COMM SMOVL C00426 BC00426 V=11.7  +MOVJ EC00426
COMM SMOVL C00427 BC00427 V=11.7  +MOVJ EC00427
COMM SFTON3D P062
COMM SMOVL C00428 BC00428 V=11.0  +MOVJ EC00428
COMM SMOVL C00429 BC00429 V=11.0  +MOVJ EC00429
COMM SFTON3D P061
COMM SMOVL C00430 BC00430 V=11.0  +MOVJ EC00430
COMM SMOVL C00431 BC00431 V=11.0  +MOVJ EC00431
COMM ARCOF
COMM SMOVL C00432 BC00432 V=800.0  +MOVJ EC00432
COMM SFTOF3D
COMM MOVJ C00433 BC00433 VJ=80.00  +MOVJ EC00433 VJ=80.00
COMM MOVJ C00434 BC00434 VJ=80.00  +MOVJ EC00434 VJ=80.00
COMM MOVJ C00435 BC00435 VJ=80.00  +MOVJ EC00435 VJ=80.00
COMM 'EndPath W3485
COMM 'Path W3486
COMM SFTOF3D
COMM SFTON3D P050
COMM MOVJ C00436 BC00436 VJ=100.00  +MOVJ EC00436 VJ=100.00
COMM SMOVL C00437 BC00437 V=800.0  +MOVJ EC00437
COMM SMOVL C00438 BC00438 V=150.0 PL=0  +MOVJ EC00438
COMM MACRO1 MJ#(0) ARGF14
COMM ARCON
COMM SMOVL C00439 BC00439 V=10.0  +MOVJ EC00439
COMM SMOVL C00440 BC00440 V=10.0  +MOVJ EC00440
COMM SMOVL C00441 BC00441 V=10.0  +MOVJ EC00441
COMM ARCOF
COMM SMOVL C00442 BC00442 V=800.0  +MOVJ EC00442
COMM SMOVL C00443 BC00443 V=1000.0  +MOVJ EC00443
COMM SFTOF3D
COMM 'EndPath W3486
COMM MOVJ C00444 BC00444 VJ=100.00  +MOVJ EC00444 VJ=100.00
COMM 'Path W3485
COMM SFTOF3D
COMM SFTON3D P034
COMM MOVJ C00445 BC00445 VJ=100.00  +MOVJ EC00445 VJ=100.00
COMM SMOVL C00446 BC00446 V=800.0  +MOVJ EC00446
COMM SMOVL C00447 BC00447 V=166.7 PL=0  +MOVJ EC00447
COMM ARCON
COMM SMOVL C00448 BC00448 V=9.2  +MOVJ EC00448
COMM SMOVL C00449 BC00449 V=9.2  +MOVJ EC00449
COMM SMOVL C00450 BC00450 V=9.2  +MOVJ EC00450
COMM ARCOF
COMM SMOVL C00451 BC00451 V=800.0  +MOVJ EC00451
COMM SMOVL C00452 BC00452 V=1000.0  +MOVJ EC00452
COMM SFTOF3D
COMM 'EndPath W3485
COMM 'Path W3487
COMM SFTOF3D
COMM SFTON3D P054
COMM MOVJ C00453 BC00453 VJ=100.00  +MOVJ EC00453 VJ=100.00
COMM SMOVL C00454 BC00454 V=800.0  +MOVJ EC00454
COMM SMOVL C00455 BC00455 V=150.0 PL=0  +MOVJ EC00455
COMM ARCON
COMM SMOVL C00456 BC00456 V=9.2  +MOVJ EC00456
COMM SMOVL C00457 BC00457 V=9.2  +MOVJ EC00457
COMM SMOVL C00458 BC00458 V=9.2  +MOVJ EC00458
COMM ARCOF
COMM SMOVL C00459 BC00459 V=800.0  +MOVJ EC00459
COMM SMOVL C00460 BC00460 V=1000.0  +MOVJ EC00460
COMM SFTOF3D
COMM 'EndPath W3487
COMM MOVJ C00461 BC00461 VJ=100.00  +MOVJ EC00461 VJ=100.00
COMM 'Path W3487
COMM SFTOF3D
COMM SFTON3D P028
COMM MOVJ C00462 BC00462 VJ=100.00  +MOVJ EC00462 VJ=100.00
COMM SMOVL C00463 BC00463 V=800.0  +MOVJ EC00463
COMM SMOVL C00464 BC00464 V=150.0 PL=0  +MOVJ EC00464
COMM ARCON
COMM SMOVL C00465 BC00465 V=9.2  +MOVJ EC00465
COMM SMOVL C00466 BC00466 V=9.2  +MOVJ EC00466
COMM SMOVL C00467 BC00467 V=9.2  +MOVJ EC00467
COMM ARCOF
COMM SMOVL C00468 BC00468 V=800.0  +MOVJ EC00468
COMM SMOVL C00469 BC00469 V=1000.0  +MOVJ EC00469
COMM SFTOF3D
COMM 'EndPath W3487
COMM MOVJ C00470 BC00470 VJ=100.00  +MOVJ EC00470 VJ=100.00
COMM MOVJ C00471 BC00471 VJ=100.00  +MOVJ EC00471 VJ=100.00
COMM 'brak dostepu offset 5mm
COMM 'Path W3488
COMM SFTOF3D
COMM SFTON3D P028
COMM MOVJ C00472 BC00472 VJ=100.00  +MOVJ EC00472 VJ=100.00
COMM SMOVL C00473 BC00473 V=800.0  +MOVJ EC00473
COMM SMOVL C00474 BC00474 V=150.0 PL=0  +MOVJ EC00474
COMM ARCON
COMM SMOVL C00475 BC00475 V=11.7  +MOVJ EC00475
COMM ARCOF
COMM SMOVL C00476 BC00476 V=800.0  +MOVJ EC00476
COMM SMOVL C00477 BC00477 V=1000.0  +MOVJ EC00477
COMM SFTOF3D
COMM 'EndPath W3488
COMM MOVJ C00478 BC00478 VJ=100.00  +MOVJ EC00478 VJ=100.00
COMM '13
COMM 'Path W3489
COMM SFTOF3D
COMM SFTON3D P030
COMM MOVJ C00479 BC00479 VJ=100.00  +MOVJ EC00479 VJ=100.00
COMM SMOVL C00480 BC00480 V=800.0  +MOVJ EC00480
COMM SMOVL C00481 BC00481 V=150.0 PL=0  +MOVJ EC00481
COMM MACRO1 MJ#(0) ARGF9
COMM ARCON
COMM SWVON WEV#(10)
COMM SFTON3D P031
COMM SMOVL C00482 BC00482 V=12.5  +MOVJ EC00482
COMM ARCOF
COMM SWVOF
COMM SMOVL C00483 BC00483 V=800.0  +MOVJ EC00483
COMM SMOVL C00484 BC00484 V=1000.0  +MOVJ EC00484
COMM SFTOF3D
COMM 'EndPath W3489
COMM 'Path W3490
COMM SFTOF3D
COMM MOVJ C00485 BC00485 VJ=100.00  +MOVJ EC00485 VJ=100.00
COMM MACRO1 MJ#(0) ARGF6
COMM SFTON3D P069
COMM SMOVL C00486 BC00486 V=250.0  +MOVJ EC00486
COMM ARCON
COMM SMOVL C00487 BC00487 V=11.7  +MOVJ EC00487
COMM ARCOF
COMM SMOVL C00488 BC00488 V=250.0  +MOVJ EC00488
COMM SFTOF3D
COMM SFTON3D P052
COMM MOVJ C00489 BC00489 VJ=100.00  +MOVJ EC00489 VJ=100.00
COMM SMOVL C00490 BC00490 V=800.0  +MOVJ EC00490
COMM SMOVL C00491 BC00491 V=150.0 PL=0  +MOVJ EC00491
COMM MACRO1 MJ#(0) ARGF14
COMM ARCON
COMM SMOVL C00492 BC00492 V=10.0  +MOVJ EC00492
COMM SMOVL C00493 BC00493 V=10.0  +MOVJ EC00493
COMM SMOVL C00494 BC00494 V=10.0  +MOVJ EC00494
COMM ARCOF
COMM SMOVL C00495 BC00495 V=800.0  +MOVJ EC00495
COMM SMOVL C00496 BC00496 V=1000.0  +MOVJ EC00496
COMM SFTOF3D
COMM 'EndPath W3490
COMM MOVJ C00497 BC00497 VJ=100.00  +MOVJ EC00497 VJ=100.00
COMM 'poprawic spoine - nie mialem w
COMM 'yciecia
COMM 'Path W3491
COMM SFTOF3D
COMM SFTON3D P053
COMM MOVJ C00498 BC00498 VJ=100.00  +MOVJ EC00498 VJ=100.00
COMM SMOVL C00499 BC00499 V=800.0  +MOVJ EC00499
COMM SMOVL C00500 BC00500 V=150.0 PL=0  +MOVJ EC00500
COMM ARCON
COMM SMOVL C00501 BC00501 V=10.0  +MOVJ EC00501
COMM SMOVL C00502 BC00502 V=10.0  +MOVJ EC00502
COMM SMOVL C00503 BC00503 V=10.0  +MOVJ EC00503
COMM ARCOF
COMM SMOVL C00504 BC00504 V=800.0  +MOVJ EC00504
COMM SMOVL C00505 BC00505 V=1000.0  +MOVJ EC00505
COMM SFTOF3D
COMM 'EndPath W3491
COMM '14
COMM '15-brak
COMM MOVJ C00506 BC00506 VJ=100.00  +MOVJ EC00506 VJ=100.00
COMM '16
COMM 'Path W3491
COMM SFTOF3D
COMM SFTON3D P029
COMM MOVJ C00507 BC00507 VJ=100.00  +MOVJ EC00507 VJ=100.00
COMM SMOVL C00508 BC00508 V=800.0  +MOVJ EC00508
COMM SMOVL C00509 BC00509 V=150.0 PL=0  +MOVJ EC00509
COMM ARCON
COMM SMOVL C00510 BC00510 V=10.0  +MOVJ EC00510
COMM SMOVL C00511 BC00511 V=10.0  +MOVJ EC00511
COMM ARCOF
COMM SMOVL C00512 BC00512 V=800.0  +MOVJ EC00512
COMM SMOVL C00513 BC00513 V=1000.0  +MOVJ EC00513
COMM SFTOF3D
COMM 'EndPath W3491
COMM MOVJ C00514 BC00514 VJ=100.00  +MOVJ EC00514 VJ=100.00
COMM 'Path W3492
COMM SFTOF3D
COMM SFTON3D P029
COMM MOVJ C00515 BC00515 VJ=100.00  +MOVJ EC00515 VJ=100.00
COMM SMOVL C00516 BC00516 V=800.0  +MOVJ EC00516
COMM SMOVL C00517 BC00517 V=150.0 PL=0  +MOVJ EC00517
COMM ARCON
COMM SMOVL C00518 BC00518 V=10.0  +MOVJ EC00518
COMM ARCOF
COMM SMOVL C00519 BC00519 V=800.0  +MOVJ EC00519
COMM SMOVL C00520 BC00520 V=1000.0  +MOVJ EC00520
COMM SFTOF3D
COMM 'EndPath W3492
COMM MOVJ C00521 BC00521 VJ=100.00  +MOVJ EC00521 VJ=100.00
COMM MOVJ C00522 BC00522 VJ=100.00  +MOVJ EC00522 VJ=100.00
COMM 'Path W3493
COMM SFTOF3D
COMM SFTON3D P029
COMM MOVJ C00523 BC00523 VJ=100.00  +MOVJ EC00523 VJ=100.00
COMM SMOVL C00524 BC00524 V=800.0  +MOVJ EC00524
COMM SMOVL C00525 BC00525 V=150.0 PL=0  +MOVJ EC00525
COMM ARCON
COMM SMOVL C00526 BC00526 V=10.0  +MOVJ EC00526
COMM SMOVL C00527 BC00527 V=10.0  +MOVJ EC00527
COMM SMOVL C00528 BC00528 V=10.0  +MOVJ EC00528
COMM ARCON
COMM SMOVL C00529 BC00529 V=11.7  +MOVJ EC00529
COMM ARCON
COMM SMOVL C00530 BC00530 V=11.7  +MOVJ EC00530
COMM ARCOF
COMM SMOVL C00531 BC00531 V=800.0  +MOVJ EC00531
COMM SMOVL C00532 BC00532 V=1000.0  +MOVJ EC00532
COMM SFTOF3D
COMM 'EndPath W3493
COMM MOVJ C00533 BC00533 VJ=100.00  +MOVJ EC00533 VJ=100.00
COMM MOVJ C00534 BC00534 VJ=100.00  +MOVJ EC00534 VJ=100.00
COMM '17
COMM 'Path W3494
COMM SFTOF3D
COMM SFTON3D P027
COMM MOVJ C00535 BC00535 VJ=100.00  +MOVJ EC00535 VJ=100.00
COMM SMOVL C00536 BC00536 V=800.0  +MOVJ EC00536
COMM SMOVL C00537 BC00537 V=150.0 PL=0  +MOVJ EC00537
COMM ARCON
COMM SMOVL C00538 BC00538 V=10.0  +MOVJ EC00538
COMM ARCOF
COMM SMOVL C00539 BC00539 V=800.0  +MOVJ EC00539
COMM SMOVL C00540 BC00540 V=1000.0  +MOVJ EC00540
COMM SFTOF3D
COMM 'EndPath W3494
COMM 'Path W3495
COMM SFTOF3D
COMM SFTON3D P027
COMM MOVJ C00541 BC00541 VJ=100.00  +MOVJ EC00541 VJ=100.00
COMM SMOVL C00542 BC00542 V=800.0  +MOVJ EC00542
COMM SMOVL C00543 BC00543 V=150.0 PL=0  +MOVJ EC00543
COMM ARCON
COMM SMOVL C00544 BC00544 V=10.8  +MOVJ EC00544
COMM ARCOF
COMM SMOVL C00545 BC00545 V=800.0  +MOVJ EC00545
COMM SMOVL C00546 BC00546 V=1000.0  +MOVJ EC00546
COMM SFTOF3D
COMM 'EndPath W3495
COMM 'Path W3496
COMM SFTOF3D
COMM SFTON3D P027
COMM MOVJ C00547 BC00547 VJ=100.00  +MOVJ EC00547 VJ=100.00
COMM SFTOF3D
COMM 'EndPath W3496
COMM MOVJ C00548 BC00548 VJ=100.00  +MOVJ EC00548 VJ=100.00
COMM MOVJ C00549 BC00549 VJ=100.00  +MOVJ EC00549 VJ=100.00
COMM MOVJ C00550 BC00550 VJ=100.00  +MOVJ EC00550 VJ=100.00
COMM '18
COMM 'Path W3497
COMM SFTOF3D
COMM SFTON3D P024
COMM MOVJ C00551 BC00551 VJ=100.00  +MOVJ EC00551 VJ=100.00
COMM SMOVL C00552 BC00552 V=800.0  +MOVJ EC00552
COMM SMOVL C00553 BC00553 V=150.0 PL=0  +MOVJ EC00553
COMM ARCON
COMM SMOVL C00554 BC00554 V=9.2  +MOVJ EC00554
COMM SMOVL C00555 BC00555 V=9.2  +MOVJ EC00555
COMM SMOVL C00556 BC00556 V=9.2  +MOVJ EC00556
COMM SMOVL C00557 BC00557 V=9.2  +MOVJ EC00557
COMM ARCOF
COMM SMOVL C00558 BC00558 V=800.0  +MOVJ EC00558
COMM SMOVL C00559 BC00559 V=1000.0  +MOVJ EC00559
COMM SFTOF3D
COMM 'EndPath W3497
COMM '
COMM 'Path W4855
COMM SFTOF3D
COMM SFTON3D P071
COMM MOVJ C00560 BC00560 VJ=100.00  +MOVJ EC00560 VJ=100.00
COMM SMOVL C00561 BC00561 V=800.0  +MOVJ EC00561
COMM MACRO1 MJ#(0) ARGF9
COMM SMOVL C00562 BC00562 V=150.0 PL=0  +MOVJ EC00562
COMM ARCON
COMM SMOVL C00563 BC00563 V=8.8  +MOVJ EC00563
COMM SFTON3D P072
COMM SMOVL C00564 BC00564 V=8.8  +MOVJ EC00564
COMM SMOVL C00565 BC00565 V=8.8  +MOVJ EC00565
COMM ARCOF
COMM SMOVL C00566 BC00566 V=800.0  +MOVJ EC00566
COMM SMOVL C00567 BC00567 V=1000.0  +MOVJ EC00567
COMM SFTOF3D
COMM 'EndPath W4855
COMM '
COMM '
COMM MOVJ C00568 BC00568 VJ=100.00  +MOVJ EC00568 VJ=100.00
COMM '19
COMM MOVJ C00569 BC00569 VJ=100.00  +MOVJ EC00569 VJ=100.00
COMM 'Path W3499
COMM SFTOF3D
COMM SFTON3D P023
COMM MOVJ C00570 BC00570 VJ=100.00  +MOVJ EC00570 VJ=100.00
COMM SMOVL C00571 BC00571 V=800.0  +MOVJ EC00571
COMM SMOVL C00572 BC00572 V=150.0 PL=0  +MOVJ EC00572
COMM MACRO1 MJ#(0) ARGF6
COMM ARCON
COMM SWVON WEV#(66)
COMM SMOVL C00573 BC00573 V=7.5  +MOVJ EC00573
COMM SMOVL C00574 BC00574 V=7.5  +MOVJ EC00574
COMM SMOVL C00575 BC00575 V=7.5  +MOVJ EC00575
COMM ARCOF
COMM SWVOF
COMM SMOVL C00576 BC00576 V=800.0  +MOVJ EC00576
COMM SMOVL C00577 BC00577 V=1000.0  +MOVJ EC00577
COMM SFTOF3D
COMM 'EndPath W3499
COMM MOVJ C00578 BC00578 VJ=100.00  +MOVJ EC00578 VJ=100.00
COMM 'Path W3500
COMM SFTOF3D
COMM SFTON3D P034
COMM MOVJ C00579 BC00579 VJ=100.00  +MOVJ EC00579 VJ=100.00
COMM SMOVL C00580 BC00580 V=800.0  +MOVJ EC00580
COMM MACRO1 MJ#(0) ARGF9
COMM SMOVL C00581 BC00581 V=150.0 PL=0  +MOVJ EC00581
COMM ARCON
COMM SMOVL C00582 BC00582 V=8.3  +MOVJ EC00582
COMM SFTON3D P050
COMM SMOVL C00583 BC00583 V=8.3  +MOVJ EC00583
COMM SMOVL C00584 BC00584 V=8.3  +MOVJ EC00584
COMM ARCOF
COMM SMOVL C00585 BC00585 V=800.0  +MOVJ EC00585
COMM SMOVL C00586 BC00586 V=1000.0  +MOVJ EC00586
COMM SFTOF3D
COMM 'EndPath W3500
COMM 'Path W3501
COMM SFTOF3D
COMM SFTON3D P051
COMM MOVJ C00587 BC00587 VJ=100.00  +MOVJ EC00587 VJ=100.00
COMM SMOVL C00588 BC00588 V=800.0  +MOVJ EC00588
COMM SMOVL C00589 BC00589 V=150.0 PL=0  +MOVJ EC00589
COMM ARCON
COMM SWVON WEV#(60)
COMM SMOVL C00590 BC00590 V=7.5  +MOVJ EC00590
COMM SMOVL C00591 BC00591 V=7.5  +MOVJ EC00591
COMM SMOVL C00592 BC00592 V=7.5  +MOVJ EC00592
COMM ARCOF
COMM SWVOF
COMM SMOVL C00593 BC00593 V=800.0  +MOVJ EC00593
COMM SMOVL C00594 BC00594 V=1000.0  +MOVJ EC00594
COMM SFTOF3D
COMM 'EndPath W3501
COMM MOVJ C00595 BC00595 VJ=100.00  +MOVJ EC00595 VJ=100.00
COMM '20
COMM MOVJ C00596 BC00596 VJ=100.00  +MOVJ EC00596 VJ=100.00
COMM MOVJ C00597 BC00597 VJ=100.00  +MOVJ EC00597 VJ=100.00
COMM 'offset 5mm
COMM 'Path W3500
COMM SFTOF3D
COMM SFTON3D P032
COMM MOVJ C00598 BC00598 VJ=100.00  +MOVJ EC00598 VJ=100.00
COMM SMOVL C00599 BC00599 V=800.0  +MOVJ EC00599
COMM SMOVL C00600 BC00600 V=150.0 PL=0  +MOVJ EC00600
COMM ARCON
COMM SMOVL C00601 BC00601 V=9.2  +MOVJ EC00601
COMM ARCOF
COMM SMOVL C00602 BC00602 V=800.0  +MOVJ EC00602
COMM SMOVL C00603 BC00603 V=1000.0  +MOVJ EC00603
COMM SFTOF3D
COMM 'EndPath W3500
COMM SFTOF3D
COMM 'EndPath W3502
COMM 'offset 5mm
COMM 'Path W3503
COMM SFTOF3D
COMM SFTON3D P032
COMM MOVJ C00604 BC00604 VJ=100.00  +MOVJ EC00604 VJ=100.00
COMM SMOVL C00605 BC00605 V=800.0  +MOVJ EC00605
COMM SMOVL C00606 BC00606 V=150.0 PL=0  +MOVJ EC00606
COMM ARCON
COMM SMOVL C00607 BC00607 V=10.0  +MOVJ EC00607
COMM ARCOF
COMM SMOVL C00608 BC00608 V=800.0  +MOVJ EC00608
COMM SMOVL C00609 BC00609 V=1000.0  +MOVJ EC00609
COMM SFTOF3D
COMM 'EndPath W3503
COMM MOVJ C00610 BC00610 VJ=100.00  +MOVJ EC00610 VJ=100.00
COMM 'Path W3504
COMM SFTOF3D
COMM SFTON3D P032
COMM MOVJ C00611 BC00611 VJ=100.00  +MOVJ EC00611 VJ=100.00
COMM SMOVL C00612 BC00612 V=800.0  +MOVJ EC00612
COMM SMOVL C00613 BC00613 V=150.0 PL=0  +MOVJ EC00613
COMM ARCON
COMM SMOVL C00614 BC00614 V=11.7  +MOVJ EC00614
COMM SMOVL C00615 BC00615 V=11.7  +MOVJ EC00615
COMM ARCOF
COMM SMOVL C00616 BC00616 V=800.0  +MOVJ EC00616
COMM SMOVL C00617 BC00617 V=1000.0  +MOVJ EC00617
COMM SFTOF3D
COMM 'EndPath W3504
COMM MOVJ C00618 BC00618 VJ=100.00  +MOVJ EC00618 VJ=100.00
COMM '21
COMM MOVJ C00619 BC00619 VJ=100.00  +MOVJ EC00619 VJ=100.00
COMM 'Path W3505
COMM SFTOF3D
COMM SFTON3D P021
COMM MOVJ C00620 BC00620 VJ=100.00  +MOVJ EC00620 VJ=100.00
COMM SMOVL C00621 BC00621 V=800.0  +MOVJ EC00621
COMM SMOVL C00622 BC00622 V=150.0 PL=0  +MOVJ EC00622
COMM ARCON
COMM SFTON3D P022
COMM SMOVL C00623 BC00623 V=10.8  +MOVJ EC00623
COMM SMOVL C00624 BC00624 V=11.7  +MOVJ EC00624
COMM ARCOF
COMM SMOVL C00625 BC00625 V=800.0  +MOVJ EC00625
COMM SMOVL C00626 BC00626 V=1000.0  +MOVJ EC00626
COMM SFTOF3D
COMM 'EndPath W3505
COMM MOVJ C00627 BC00627 VJ=100.00  +MOVJ EC00627 VJ=100.00
COMM 'Path W3506
COMM SFTOF3D
COMM SFTON3D P095
COMM MOVJ C00628 BC00628 VJ=100.00  +MOVJ EC00628 VJ=100.00
COMM SMOVL C00629 BC00629 V=800.0  +MOVJ EC00629
COMM SMOVL C00630 BC00630 V=150.0 PL=0  +MOVJ EC00630
COMM MACRO1 MJ#(0) ARGF14
COMM ARCON
COMM SMOVL C00631 BC00631 V=10.0  +MOVJ EC00631
COMM SMOVL C00632 BC00632 V=10.0  +MOVJ EC00632
COMM SMOVL C00633 BC00633 V=10.0  +MOVJ EC00633
COMM ARCOF
COMM SMOVL C00634 BC00634 V=800.0  +MOVJ EC00634
COMM SMOVL C00635 BC00635 V=1000.0  +MOVJ EC00635
COMM SFTOF3D
COMM 'EndPath W3506
COMM 'Path W3507
COMM SFTOF3D
COMM SFTON3D P096
COMM MOVJ C00636 BC00636 VJ=100.00  +MOVJ EC00636 VJ=100.00
COMM SMOVL C00637 BC00637 V=800.0  +MOVJ EC00637
COMM SMOVL C00638 BC00638 V=150.0 PL=0  +MOVJ EC00638
COMM ARCON
COMM SMOVL C00639 BC00639 V=10.0  +MOVJ EC00639
COMM SMOVL C00640 BC00640 V=10.0  +MOVJ EC00640
COMM ARCOF
COMM SMOVL C00641 BC00641 V=800.0  +MOVJ EC00641
COMM SMOVL C00642 BC00642 V=1000.0  +MOVJ EC00642
COMM SFTOF3D
COMM 'EndPath W3507
COMM MOVJ C00643 BC00643 VJ=100.00  +MOVJ EC00643 VJ=100.00
COMM MOVJ C00644 BC00644 VJ=100.00  +MOVJ EC00644 VJ=100.00
COMM 'Path W4856
COMM SFTOF3D
COMM SFTON3D P071
COMM MOVJ C00645 BC00645 VJ=100.00  +MOVJ EC00645 VJ=100.00
COMM SMOVL C00646 BC00646 V=800.0  +MOVJ EC00646
COMM SMOVL C00647 BC00647 V=150.0 PL=0  +MOVJ EC00647
COMM ARCON
COMM SMOVL C00648 BC00648 V=8.3  +MOVJ EC00648
COMM SFTON3D P073
COMM SMOVL C00649 BC00649 V=8.3  +MOVJ EC00649
COMM SMOVL C00650 BC00650 V=8.3  +MOVJ EC00650
COMM ARCOF
COMM SMOVL C00651 BC00651 V=800.0  +MOVJ EC00651
COMM SMOVL C00652 BC00652 V=1000.0  +MOVJ EC00652
COMM SFTOF3D
COMM 'EndPath W4856
COMM MOVJ C00653 BC00653 VJ=100.00  +MOVJ EC00653 VJ=100.00
COMM MOVJ C00654 BC00654 VJ=100.00  +MOVJ EC00654 VJ=100.00
'X2_8A-21A(90,0)
MOVJ C00655 BC00655 VJ=100.00  +MOVJ EC00655 VJ=100.00
CALL JOB:CLEAN-R1_KM_3P
MOVJ C00656 BC00656 VJ=100.00  +MOVJ EC00656 VJ=100.00
MOVJ C00657 BC00657 VJ=100.00  +MOVJ EC00657 VJ=100.00
'Path S3463
SFTOF3D
MOVJ C00658 BC00658 VJ=100.00  +MOVJ EC00658 VJ=100.00
MOVL C00659 BC00659 V=666.7  +MOVJ EC00659 VJ=100.00
SMOVL C00660 BC00660 V=166.7  +MOVJ EC00660
SREFP 3 C00661 BC00661  +REFP EC00661
CALL JOB:SEARCH-R1-S13D
SET P095 P006
SFTON3D P095
SMOVL C00662 BC00662 V=166.7  +MOVJ EC00662
SMOVL C00663 BC00663 V=166.7  +MOVJ EC00663
SREFP 3 C00664 BC00664  +REFP EC00664
CALL JOB:SEARCH-R1-S13D
SET P095 P006
SFTON3D P095
SMOVL C00665 BC00665 V=166.7  +MOVJ EC00665
MOVL C00666 BC00666 V=1000.0  +MOVJ EC00666 VJ=100.00
'EndPath S3463
'Path S3464
SFTOF3D
MOVJ C00667 BC00667 VJ=100.00  +MOVJ EC00667 VJ=100.00
MOVL C00668 BC00668 V=666.7  +MOVJ EC00668 VJ=100.00
SMOVL C00669 BC00669 V=166.7  +MOVJ EC00669
SREFP 3 C00670 BC00670  +REFP EC00670
CALL JOB:SEARCH-R1-S13D
SET P096 P006
SFTON3D P096
SMOVL C00671 BC00671 V=166.7  +MOVJ EC00671
SREFP 3 C00672 BC00672  +REFP EC00672
CALL JOB:SEARCH-R1-S13D
SET P096 P006
SFTON3D P096
SMOVL C00673 BC00673 V=166.7  +MOVJ EC00673
MOVL C00674 BC00674 V=1000.0  +MOVJ EC00674 VJ=100.00
'EndPath S3464
'Path S3465
SFTOF3D
MOVJ C00675 BC00675 VJ=100.00  +MOVJ EC00675 VJ=100.00
MOVL C00676 BC00676 V=666.7  +MOVJ EC00676 VJ=100.00
MOVL C00677 BC00677 V=666.7  +MOVJ EC00677 VJ=100.00
SMOVL C00678 BC00678 V=166.7  +MOVJ EC00678
SREFP 3 C00679 BC00679  +REFP EC00679
CALL JOB:SEARCH-R1-S13D
SET P097 P006
SFTON3D P097
SMOVL C00680 BC00680 V=166.7  +MOVJ EC00680
SMOVL C00681 BC00681 V=166.7  +MOVJ EC00681
SREFP 3 C00682 BC00682  +REFP EC00682
CALL JOB:SEARCH-R1-S13D
SET P097 P006
SFTON3D P097
SMOVL C00683 BC00683 V=166.7  +MOVJ EC00683
SMOVL C00684 BC00684 V=166.7  +MOVJ EC00684
SREFP 3 C00685 BC00685  +REFP EC00685
CALL JOB:SEARCH-R1-S13D
SET P021 P006
SFTON3D P021
SMOVL C00686 BC00686 V=166.7  +MOVJ EC00686
SMOVL C00687 BC00687 V=166.7  +MOVJ EC00687
SREFP 3 C00688 BC00688  +REFP EC00688
CALL JOB:SEARCH-R1-S13D
SET P021 P006
SFTON3D P021
SMOVL C00689 BC00689 V=166.7  +MOVJ EC00689
MOVL C00690 BC00690 V=1000.0  +MOVJ EC00690 VJ=100.00
'EndPath S3465
'Path S3464
SFTOF3D
MOVJ C00691 BC00691 VJ=100.00  +MOVJ EC00691 VJ=100.00
MOVL C00692 BC00692 V=666.7  +MOVJ EC00692 VJ=100.00
SMOVL C00693 BC00693 V=166.7  +MOVJ EC00693
SREFP 3 C00694 BC00694  +REFP EC00694
CALL JOB:SEARCH-R1-S13D
SET P022 P006
SFTON3D P022
SMOVL C00695 BC00695 V=166.7  +MOVJ EC00695
SREFP 3 C00696 BC00696  +REFP EC00696
CALL JOB:SEARCH-R1-S13D
SET P022 P006
SFTON3D P022
SMOVL C00697 BC00697 V=166.7  +MOVJ EC00697
MOVL C00698 BC00698 V=1000.0  +MOVJ EC00698 VJ=100.00
'EndPath S3464
MOVJ C00699 BC00699 VJ=100.00  +MOVJ EC00699 VJ=100.00
'Path S3465
SFTOF3D
MOVJ C00700 BC00700 VJ=100.00  +MOVJ EC00700 VJ=100.00
MOVL C00701 BC00701 V=666.7  +MOVJ EC00701 VJ=100.00
SMOVL C00702 BC00702 V=166.7  +MOVJ EC00702
SREFP 3 C00703 BC00703  +REFP EC00703
CALL JOB:SEARCH-R1-S13D
SET P050 P006
SFTON3D P050
SMOVL C00704 BC00704 V=166.7  +MOVJ EC00704
SREFP 3 C00705 BC00705  +REFP EC00705
CALL JOB:SEARCH-R1-S13D
SET P050 P006
SFTON3D P050
SMOVL C00706 BC00706 V=166.7  +MOVJ EC00706
SMOVL C00707 BC00707 V=166.7  +MOVJ EC00707
SREFP 3 C00708 BC00708  +REFP EC00708
CALL JOB:SEARCH-R1-S13D
SET P050 P006
SFTON3D P050
SMOVL C00709 BC00709 V=166.7  +MOVJ EC00709
MOVL C00710 BC00710 V=1000.0  +MOVJ EC00710 VJ=100.00
'EndPath S3465
'Path S3466
SFTOF3D
MOVJ C00711 BC00711 VJ=100.00  +MOVJ EC00711 VJ=100.00
MOVL C00712 BC00712 V=666.7  +MOVJ EC00712 VJ=100.00
SMOVL C00713 BC00713 V=166.7  +MOVJ EC00713
SREFP 3 C00714 BC00714  +REFP EC00714
CALL JOB:SEARCH-R1-S13D
SET P051 P006
SFTON3D P051
SMOVL C00715 BC00715 V=166.7  +MOVJ EC00715
SREFP 3 C00716 BC00716  +REFP EC00716
CALL JOB:SEARCH-R1-S13D
SET P051 P006
SFTON3D P051
SMOVL C00717 BC00717 V=166.7  +MOVJ EC00717
SMOVL C00718 BC00718 V=250.0  +MOVJ EC00718
SREFP 3 C00719 BC00719  +REFP EC00719
CALL JOB:SEARCH-R1-S13D
SET P051 P006
SFTON3D P051
SMOVL C00720 BC00720 V=166.7  +MOVJ EC00720
MOVL C00721 BC00721 V=1000.0  +MOVJ EC00721 VJ=100.00
'EndPath S3466
MOVJ C00722 BC00722 VJ=100.00  +MOVJ EC00722 VJ=100.00
MOVJ C00723 BC00723 VJ=100.00  +MOVJ EC00723 VJ=100.00
'Path S3467
SFTOF3D
MOVJ C00724 BC00724 VJ=100.00  +MOVJ EC00724 VJ=100.00
MOVL C00725 BC00725 V=666.7  +MOVJ EC00725 VJ=100.00
SMOVL C00726 BC00726 V=166.7  +MOVJ EC00726
SREFP 3 C00727 BC00727  +REFP EC00727
CALL JOB:SEARCH-R1-S13D
SET P054 P006
SFTON3D P054
SMOVL C00728 BC00728 V=250.0  +MOVJ EC00728
SMOVL C00729 BC00729 V=166.7  +MOVJ EC00729
SREFP 3 C00730 BC00730  +REFP EC00730
CALL JOB:SEARCH-R1-S13D
SET P054 P006
SFTON3D P054
SMOVL C00731 BC00731 V=166.7  +MOVJ EC00731
SMOVL C00732 BC00732 V=800.0  +MOVJ EC00732
SMOVL C00733 BC00733 V=166.7  +MOVJ EC00733
SREFP 3 C00734 BC00734  +REFP EC00734
CALL JOB:SEARCH-R1-S13D
SET P054 P006
SFTON3D P054
SMOVL C00735 BC00735 V=166.7  +MOVJ EC00735
MOVL C00736 BC00736 V=1000.0  +MOVJ EC00736 VJ=100.00
'EndPath S3467
'Path S3475
SFTOF3D
MOVJ C00737 BC00737 VJ=100.00  +MOVJ EC00737 VJ=100.00
MOVL C00738 BC00738 V=666.7  +MOVJ EC00738 VJ=100.00
SMOVL C00739 BC00739 V=166.7  +MOVJ EC00739
SREFP 3 C00740 BC00740  +REFP EC00740
CALL JOB:SEARCH-R1-S13D
SET P034 P006
SFTON3D P034
SMOVL C00741 BC00741 V=166.7  +MOVJ EC00741
SMOVL C00742 BC00742 V=333.3  +MOVJ EC00742
SMOVL C00743 BC00743 V=166.7  +MOVJ EC00743
SREFP 3 C00744 BC00744  +REFP EC00744
CALL JOB:SEARCH-R1-S13D
SET P034 P006
SFTON3D P034
SMOVL C00745 BC00745 V=166.7  +MOVJ EC00745
SMOVL C00746 BC00746 V=166.7  +MOVJ EC00746
SREFP 3 C00747 BC00747  +REFP EC00747
CALL JOB:SEARCH-R1-S13D
SET P034 P006
SFTON3D P034
SMOVL C00748 BC00748 V=166.7  +MOVJ EC00748
MOVL C00749 BC00749 V=1000.0  +MOVJ EC00749 VJ=100.00
'EndPath S3475
'Path S3464
SFTOF3D
MOVJ C00750 BC00750 VJ=100.00  +MOVJ EC00750 VJ=100.00
MOVL C00751 BC00751 V=666.7  +MOVJ EC00751 VJ=100.00
SMOVL C00752 BC00752 V=166.7  +MOVJ EC00752
SREFP 3 C00753 BC00753  +REFP EC00753
CALL JOB:SEARCH-R1-S13D
SET P023 P006
SFTON3D P023
SMOVL C00754 BC00754 V=166.7  +MOVJ EC00754
SMOVL C00755 BC00755 V=500.0  +MOVJ EC00755
SMOVL C00756 BC00756 V=166.7  +MOVJ EC00756
SREFP 3 C00757 BC00757  +REFP EC00757
CALL JOB:SEARCH-R1-S13D
SET P023 P006
SFTON3D P023
SMOVL C00758 BC00758 V=166.7  +MOVJ EC00758
SMOVL C00759 BC00759 V=166.7  +MOVJ EC00759
SREFP 3 C00760 BC00760  +REFP EC00760
CALL JOB:SEARCH-R1-S13D
SET P023 P006
SFTON3D P023
SMOVL C00761 BC00761 V=166.7  +MOVJ EC00761
MOVL C00762 BC00762 V=1000.0  +MOVJ EC00762 VJ=100.00
MOVJ C00763 BC00763 VJ=80.00  +MOVJ EC00763 VJ=80.00
MOVJ C00764 BC00764 VJ=80.00  +MOVJ EC00764 VJ=80.00
SFTOF3D
MOVJ C00765 BC00765 VJ=80.00  +MOVJ EC00765 VJ=80.00
SMOVL C00766 BC00766 V=166.7  +MOVJ EC00766
SREFP 3 C00767 BC00767  +REFP EC00767
CALL JOB:SEARCH-R1-S13D
SET P061 P006
SFTON3D P061
SMOVL C00768 BC00768 V=166.7  +MOVJ EC00768
SREFP 3 C00769 BC00769  +REFP EC00769
CALL JOB:SEARCH-R1-S13D
SET P061 P006
SFTON3D P061
SMOVL C00770 BC00770 V=166.7  +MOVJ EC00770
SFTOF3D
SMOVL C00771 BC00771 V=500.0  +MOVJ EC00771
SMOVL C00772 BC00772 V=166.7  +MOVJ EC00772
SREFP 3 C00773 BC00773  +REFP EC00773
CALL JOB:SEARCH-R1-S13D
SET P062 P006
SFTON3D P062
SMOVL C00774 BC00774 V=166.7  +MOVJ EC00774
SREFP 3 C00775 BC00775  +REFP EC00775
CALL JOB:SEARCH-R1-S13D
SET P062 P006
SFTON3D P062
SMOVL C00776 BC00776 V=166.7  +MOVJ EC00776
SFTOF3D
SMOVL C00777 BC00777 V=500.0  +MOVJ EC00777
SMOVL C00778 BC00778 V=166.7  +MOVJ EC00778
SREFP 3 C00779 BC00779  +REFP EC00779
CALL JOB:SEARCH-R1-S13D
SET P063 P006
SFTON3D P063
SMOVL C00780 BC00780 V=166.7  +MOVJ EC00780
SREFP 3 C00781 BC00781  +REFP EC00781
CALL JOB:SEARCH-R1-S13D
SET P063 P006
SFTON3D P063
SMOVL C00782 BC00782 V=166.7  +MOVJ EC00782
SFTOF3D
SMOVL C00783 BC00783 V=500.0  +MOVJ EC00783
MOVJ C00784 BC00784 VJ=80.00  +MOVJ EC00784 VJ=80.00
MOVJ C00785 BC00785 VJ=80.00  +MOVJ EC00785 VJ=80.00
'EndPath S3464
MOVJ C00786 BC00786 VJ=100.00  +MOVJ EC00786 VJ=100.00
'Path S3465
SFTOF3D
MOVJ C00787 BC00787 VJ=100.00  +MOVJ EC00787 VJ=100.00
MOVL C00788 BC00788 V=666.7  +MOVJ EC00788 VJ=100.00
SMOVL C00789 BC00789 V=166.7  +MOVJ EC00789
SREFP 3 C00790 BC00790  +REFP EC00790
CALL JOB:SEARCH-R1-S13D
SET P024 P006
SFTON3D P024
SMOVL C00791 BC00791 V=166.7  +MOVJ EC00791
SREFP 3 C00792 BC00792  +REFP EC00792
CALL JOB:SEARCH-R1-S13D
SET P024 P006
SFTON3D P024
SMOVL C00793 BC00793 V=166.7  +MOVJ EC00793
SMOVL C00794 BC00794 V=166.7  +MOVJ EC00794
SREFP 3 C00795 BC00795  +REFP EC00795
CALL JOB:SEARCH-R1-S13D
SET P024 P006
SFTON3D P024
SMOVL C00796 BC00796 V=166.7  +MOVJ EC00796
MOVL C00797 BC00797 V=1000.0  +MOVJ EC00797 VJ=100.00
'EndPath S3465
'Path S3476
SFTOF3D
MOVJ C00798 BC00798 VJ=100.00  +MOVJ EC00798 VJ=100.00
MOVL C00799 BC00799 V=666.7  +MOVJ EC00799 VJ=100.00
SMOVL C00800 BC00800 V=166.7  +MOVJ EC00800
SREFP 3 C00801 BC00801  +REFP EC00801
CALL JOB:SEARCH-R1-S13D
SET P035 P006
SFTON3D P035
SMOVL C00802 BC00802 V=166.7  +MOVJ EC00802
SREFP 3 C00803 BC00803  +REFP EC00803
CALL JOB:SEARCH-R1-S13D
SET P035 P006
SFTON3D P035
SMOVL C00804 BC00804 V=166.7  +MOVJ EC00804
SMOVL C00805 BC00805 V=333.3  +MOVJ EC00805
SMOVL C00806 BC00806 V=166.7  +MOVJ EC00806
SREFP 3 C00807 BC00807  +REFP EC00807
CALL JOB:SEARCH-R1-S13D
SET P035 P006
SFTON3D P035
SMOVL C00808 BC00808 V=166.7  +MOVJ EC00808
MOVL C00809 BC00809 V=1000.0  +MOVJ EC00809 VJ=100.00
'EndPath S3476
'Path S3470
SFTOF3D
MOVJ C00810 BC00810 VJ=100.00  +MOVJ EC00810 VJ=100.00
MOVL C00811 BC00811 V=666.7  +MOVJ EC00811 VJ=100.00
SMOVL C00812 BC00812 V=166.7  +MOVJ EC00812
SREFP 3 C00813 BC00813  +REFP EC00813
CALL JOB:SEARCH-R1-S13D
SET P029 P006
SFTON3D P029
SMOVL C00814 BC00814 V=166.7  +MOVJ EC00814
SREFP 3 C00815 BC00815  +REFP EC00815
CALL JOB:SEARCH-R1-S13D
SET P029 P006
SFTON3D P029
SMOVL C00816 BC00816 V=166.7  +MOVJ EC00816
SMOVL C00817 BC00817 V=250.0  +MOVJ EC00817
SMOVL C00818 BC00818 V=166.7  +MOVJ EC00818
SREFP 3 C00819 BC00819  +REFP EC00819
CALL JOB:SEARCH-R1-S13D
SET P029 P006
SFTON3D P029
SMOVL C00820 BC00820 V=166.7  +MOVJ EC00820
MOVL C00821 BC00821 V=1000.0  +MOVJ EC00821 VJ=100.00
'EndPath S3470
'Path S4850
SFTOF3D
MOVL C00822 BC00822 V=666.7  +MOVJ EC00822 VJ=100.00
SMOVL C00823 BC00823 V=166.7  +MOVJ EC00823
SREFP 3 C00824 BC00824  +REFP EC00824
CALL JOB:SEARCH-R1-S13D
SET P071 P006
SFTON3D P071
SMOVL C00825 BC00825 V=166.7  +MOVJ EC00825
SREFP 3 C00826 BC00826  +REFP EC00826
CALL JOB:SEARCH-R1-S13D
SET P071 P006
SFTON3D P071
SMOVL C00827 BC00827 V=166.7  +MOVJ EC00827
SMOVL C00828 BC00828 V=166.7  +MOVJ EC00828
SREFP 3 C00829 BC00829  +REFP EC00829
CALL JOB:SEARCH-R1-S13D
SET P071 P006
SFTON3D P071
SMOVL C00830 BC00830 V=166.7  +MOVJ EC00830
MOVL C00831 BC00831 V=1000.0  +MOVJ EC00831 VJ=100.00
'EndPath S4850
'Path S4851
SFTOF3D
MOVJ C00832 BC00832 VJ=100.00  +MOVJ EC00832 VJ=100.00
'POMIAR_DOD_WZM_BOK
MOVL C00833 BC00833 V=666.7  +MOVJ EC00833 VJ=100.00
SMOVL C00834 BC00834 V=166.7  +MOVJ EC00834
SREFP 3 C00835 BC00835  +REFP EC00835
CALL JOB:SEARCH-R1-S13D
SET P080 P006
SFTON3D P080
SMOVL C00836 BC00836 V=166.7  +MOVJ EC00836
SREFP 3 C00837 BC00837  +REFP EC00837
CALL JOB:SEARCH-R1-S13D
SET P080 P006
SFTON3D P080
SMOVL C00838 BC00838 V=166.7  +MOVJ EC00838
SMOVL C00839 BC00839 V=250.0  +MOVJ EC00839
SMOVL C00840 BC00840 V=166.7  +MOVJ EC00840
SREFP 3 C00841 BC00841  +REFP EC00841
CALL JOB:SEARCH-R1-S13D
SET P080 P006
SFTON3D P080
SMOVL C00842 BC00842 V=166.7  +MOVJ EC00842
MOVL C00843 BC00843 V=1000.0  +MOVJ EC00843 VJ=100.00
SFTOF3D
MOVJ C00844 BC00844 VJ=100.00  +MOVJ EC00844 VJ=100.00
MOVL C00845 BC00845 V=666.7  +MOVJ EC00845 VJ=100.00
SMOVL C00846 BC00846 V=166.7  +MOVJ EC00846
SREFP 3 C00847 BC00847  +REFP EC00847
CALL JOB:SEARCH-R1-S13D
SET P072 P006
SFTON3D P072
SMOVL C00848 BC00848 V=166.7  +MOVJ EC00848
SREFP 3 C00849 BC00849  +REFP EC00849
CALL JOB:SEARCH-R1-S13D
SET P072 P006
SFTON3D P072
SMOVL C00850 BC00850 V=166.7  +MOVJ EC00850
MOVL C00851 BC00851 V=1000.0  +MOVJ EC00851 VJ=100.00
'EndPath S4851
MOVJ C00852 BC00852 VJ=100.00  +MOVJ EC00852 VJ=100.00
MOVJ C00853 BC00853 VJ=100.00  +MOVJ EC00853 VJ=100.00
'Path S4852
SFTOF3D
MOVJ C00854 BC00854 VJ=100.00  +MOVJ EC00854 VJ=100.00
MOVL C00855 BC00855 V=666.7  +MOVJ EC00855 VJ=100.00
SMOVL C00856 BC00856 V=166.7  +MOVJ EC00856
SREFP 3 C00857 BC00857  +REFP EC00857
CALL JOB:SEARCH-R1-S13D
SET P073 P006
SFTON3D P073
SMOVL C00858 BC00858 V=166.7  +MOVJ EC00858
SMOVL C00859 BC00859 V=166.7  +MOVJ EC00859
SREFP 3 C00860 BC00860  +REFP EC00860
CALL JOB:SEARCH-R1-S13D
SET P073 P006
SFTON3D P073
SMOVL C00861 BC00861 V=166.7  +MOVJ EC00861
SMOVL C00862 BC00862 V=166.7  +MOVJ EC00862
SREFP 3 C00863 BC00863  +REFP EC00863
CALL JOB:SEARCH-R1-S13D
SET P073 P006
SFTON3D P073
SMOVL C00864 BC00864 V=166.7  +MOVJ EC00864
MOVL C00865 BC00865 V=1000.0  +MOVJ EC00865 VJ=100.00
'EndPath S4852
MOVJ C00866 BC00866 VJ=100.00  +MOVJ EC00866 VJ=100.00
'Path S4853
SFTOF3D
MOVJ C00867 BC00867 VJ=100.00  +MOVJ EC00867 VJ=100.00
MOVL C00868 BC00868 V=666.7  +MOVJ EC00868 VJ=100.00
SMOVL C00869 BC00869 V=166.7  +MOVJ EC00869
SREFP 3 C00870 BC00870  +REFP EC00870
CALL JOB:SEARCH-R1-S13D
SET P074 P006
SFTON3D P074
SMOVL C00871 BC00871 V=166.7  +MOVJ EC00871
SREFP 3 C00872 BC00872  +REFP EC00872
CALL JOB:SEARCH-R1-S13D
SET P074 P006
SFTON3D P074
SMOVL C00873 BC00873 V=166.7  +MOVJ EC00873
MOVL C00874 BC00874 V=1000.0  +MOVJ EC00874 VJ=100.00
'EndPath S4853
'Path S3467
SFTOF3D
MOVJ C00875 BC00875 VJ=100.00  +MOVJ EC00875 VJ=100.00
MOVJ C00876 BC00876 VJ=100.00  +MOVJ EC00876 VJ=100.00
MOVL C00877 BC00877 V=666.7  +MOVJ EC00877 VJ=100.00
SMOVL C00878 BC00878 V=166.7  +MOVJ EC00878
SREFP 3 C00879 BC00879  +REFP EC00879
CALL JOB:SEARCH-R1-S13D
SET P081 P006
SFTON3D P081
SMOVL C00880 BC00880 V=166.7  +MOVJ EC00880
SMOVL C00881 BC00881 V=166.7  +MOVJ EC00881
SREFP 3 C00882 BC00882  +REFP EC00882
CALL JOB:SEARCH-R1-S13D
SET P081 P006
SFTON3D P081
SMOVL C00883 BC00883 V=166.7  +MOVJ EC00883
SMOVL C00884 BC00884 V=800.0  +MOVJ EC00884
SMOVL C00885 BC00885 V=166.7  +MOVJ EC00885
SREFP 3 C00886 BC00886  +REFP EC00886
CALL JOB:SEARCH-R1-S13D
SET P081 P006
SFTON3D P081
SMOVL C00887 BC00887 V=166.7  +MOVJ EC00887
MOVJ C00888 BC00888 VJ=100.00  +MOVJ EC00888 VJ=100.00
MOVJ C00889 BC00889 VJ=100.00  +MOVJ EC00889 VJ=100.00
SFTOF3D
MOVJ C00890 BC00890 VJ=100.00  +MOVJ EC00890 VJ=100.00
MOVL C00891 BC00891 V=666.7  +MOVJ EC00891 VJ=100.00
SMOVL C00892 BC00892 V=166.7  +MOVJ EC00892
SREFP 3 C00893 BC00893  +REFP EC00893
CALL JOB:SEARCH-R1-S13D
SET P026 P006
SFTON3D P026
SMOVL C00894 BC00894 V=166.7  +MOVJ EC00894
SREFP 3 C00895 BC00895  +REFP EC00895
CALL JOB:SEARCH-R1-S13D
SET P026 P006
SFTON3D P026
SMOVL C00896 BC00896 V=166.7  +MOVJ EC00896
SMOVL C00897 BC00897 V=800.0  +MOVJ EC00897
SMOVL C00898 BC00898 V=166.7  +MOVJ EC00898
SREFP 3 C00899 BC00899  +REFP EC00899
CALL JOB:SEARCH-R1-S13D
SET P026 P006
SFTON3D P026
SMOVL C00900 BC00900 V=166.7  +MOVJ EC00900
MOVL C00901 BC00901 V=1000.0  +MOVJ EC00901 VJ=100.00
'EndPath S3467
MOVJ C00902 BC00902 VJ=100.00  +MOVJ EC00902 VJ=100.00
'Path S3466
SFTOF3D
MOVJ C00903 BC00903 VJ=100.00  +MOVJ EC00903 VJ=100.00
MOVL C00904 BC00904 V=666.7  +MOVJ EC00904 VJ=100.00
SMOVL C00905 BC00905 V=166.7  +MOVJ EC00905
SREFP 3 C00906 BC00906  +REFP EC00906
CALL JOB:SEARCH-R1-S13D
SET P025 P006
SFTON3D P025
SMOVL C00907 BC00907 V=166.7  +MOVJ EC00907
SMOVL C00908 BC00908 V=166.7  +MOVJ EC00908
SREFP 3 C00909 BC00909  +REFP EC00909
CALL JOB:SEARCH-R1-S13D
SET P025 P006
SFTON3D P025
SMOVL C00910 BC00910 V=166.7  +MOVJ EC00910
SMOVL C00911 BC00911 V=200.0  +MOVJ EC00911
SMOVL C00912 BC00912 V=166.7  +MOVJ EC00912
SREFP 3 C00913 BC00913  +REFP EC00913
CALL JOB:SEARCH-R1-S13D
SET P025 P006
SFTON3D P025
SMOVL C00914 BC00914 V=166.7  +MOVJ EC00914
MOVL C00915 BC00915 V=1000.0  +MOVJ EC00915 VJ=100.00
'EndPath S3466
MOVJ C00916 BC00916 VJ=100.00  +MOVJ EC00916 VJ=100.00
'Path S3469
SFTOF3D
MOVJ C00917 BC00917 VJ=100.00  +MOVJ EC00917 VJ=100.00
MOVL C00918 BC00918 V=666.7  +MOVJ EC00918 VJ=100.00
SMOVL C00919 BC00919 V=166.7  +MOVJ EC00919
SREFP 3 C00920 BC00920  +REFP EC00920
CALL JOB:SEARCH-R1-S13D
SET P028 P006
SFTON3D P028
SMOVL C00921 BC00921 V=166.7  +MOVJ EC00921
SREFP 3 C00922 BC00922  +REFP EC00922
CALL JOB:SEARCH-R1-S13D
SET P028 P006
SFTON3D P028
SMOVL C00923 BC00923 V=166.7  +MOVJ EC00923
SMOVL C00924 BC00924 V=333.3  +MOVJ EC00924
SMOVL C00925 BC00925 V=166.7  +MOVJ EC00925
SREFP 3 C00926 BC00926  +REFP EC00926
CALL JOB:SEARCH-R1-S13D
SET P028 P006
SFTON3D P028
SMOVL C00927 BC00927 V=166.7  +MOVJ EC00927
MOVL C00928 BC00928 V=1000.0  +MOVJ EC00928 VJ=100.00
'EndPath S3469
MOVJ C00929 BC00929 VJ=100.00  +MOVJ EC00929 VJ=100.00
'Path S3474
SFTOF3D
MOVJ C00930 BC00930 VJ=100.00  +MOVJ EC00930 VJ=100.00
MOVL C00931 BC00931 V=666.7  +MOVJ EC00931 VJ=100.00
SMOVL C00932 BC00932 V=166.7  +MOVJ EC00932
SREFP 3 C00933 BC00933  +REFP EC00933
CALL JOB:SEARCH-R1-S13D
SET P033 P006
SFTON3D P033
SMOVL C00934 BC00934 V=166.7  +MOVJ EC00934
SREFP 3 C00935 BC00935  +REFP EC00935
CALL JOB:SEARCH-R1-S13D
SET P033 P006
SFTON3D P033
SMOVL C00936 BC00936 V=166.7  +MOVJ EC00936
SMOVL C00937 BC00937 V=250.0  +MOVJ EC00937
SMOVL C00938 BC00938 V=166.7  +MOVJ EC00938
SREFP 3 C00939 BC00939  +REFP EC00939
CALL JOB:SEARCH-R1-S13D
SET P033 P006
SFTON3D P033
SMOVL C00940 BC00940 V=166.7  +MOVJ EC00940
MOVL C00941 BC00941 V=1000.0  +MOVJ EC00941 VJ=100.00
'EndPath S3474
'Path S3468
SFTOF3D
MOVJ C00942 BC00942 VJ=100.00  +MOVJ EC00942 VJ=100.00
MOVL C00943 BC00943 V=666.7  +MOVJ EC00943 VJ=100.00
SMOVL C00944 BC00944 V=166.7  +MOVJ EC00944
SREFP 3 C00945 BC00945  +REFP EC00945
CALL JOB:SEARCH-R1-S13D
SET P027 P006
SFTON3D P027
SMOVL C00946 BC00946 V=166.7  +MOVJ EC00946
SMOVL C00947 BC00947 V=166.7  +MOVJ EC00947
SREFP 3 C00948 BC00948  +REFP EC00948
CALL JOB:SEARCH-R1-S13D
SET P027 P006
SFTON3D P027
SMOVL C00949 BC00949 V=166.7  +MOVJ EC00949
SMOVL C00950 BC00950 V=166.7  +MOVJ EC00950
SREFP 3 C00951 BC00951  +REFP EC00951
CALL JOB:SEARCH-R1-S13D
SET P027 P006
SFTON3D P027
SMOVL C00952 BC00952 V=166.7  +MOVJ EC00952
MOVL C00953 BC00953 V=1000.0  +MOVJ EC00953 VJ=100.00
'EndPath S3468
'Path S3471
SFTOF3D
MOVJ C00954 BC00954 VJ=100.00  +MOVJ EC00954 VJ=100.00
MOVL C00955 BC00955 V=666.7  +MOVJ EC00955 VJ=100.00
SMOVL C00956 BC00956 V=166.7  +MOVJ EC00956
SREFP 3 C00957 BC00957  +REFP EC00957
CALL JOB:SEARCH-R1-S13D
SET P030 P006
SFTON3D P030
SMOVL C00958 BC00958 V=166.7  +MOVJ EC00958
SREFP 3 C00959 BC00959  +REFP EC00959
CALL JOB:SEARCH-R1-S13D
SET P030 P006
SFTON3D P030
SMOVL C00960 BC00960 V=166.7  +MOVJ EC00960
MOVL C00961 BC00961 V=1000.0  +MOVJ EC00961 VJ=100.00
'EndPath S3471
'Path S3472
SFTOF3D
MOVJ C00962 BC00962 VJ=100.00  +MOVJ EC00962 VJ=100.00
MOVL C00963 BC00963 V=666.7  +MOVJ EC00963 VJ=100.00
SMOVL C00964 BC00964 V=166.7  +MOVJ EC00964
SREFP 3 C00965 BC00965  +REFP EC00965
CALL JOB:SEARCH-R1-S13D
SET P031 P006
SFTON3D P031
SMOVL C00966 BC00966 V=166.7  +MOVJ EC00966
SREFP 3 C00967 BC00967  +REFP EC00967
CALL JOB:SEARCH-R1-S13D
SET P031 P006
SFTON3D P031
SMOVL C00968 BC00968 V=166.7  +MOVJ EC00968
MOVL C00969 BC00969 V=1000.0  +MOVJ EC00969 VJ=100.00
MOVL C00970 BC00970 V=666.7  +MOVJ EC00970 VJ=100.00
SMOVL C00971 BC00971 V=166.7  +MOVJ EC00971
SREFP 3 C00972 BC00972  +REFP EC00972
CALL JOB:SEARCH-R1-S13D
SET P098 P006
SFTON3D P098
SMOVL C00973 BC00973 V=166.7  +MOVJ EC00973
SREFP 3 C00974 BC00974  +REFP EC00974
CALL JOB:SEARCH-R1-S13D
SET P098 P006
SFTON3D P098
SMOVL C00975 BC00975 V=166.7  +MOVJ EC00975
MOVL C00976 BC00976 V=1000.0  +MOVJ EC00976 VJ=100.00
'EndPath S3472
MOVJ C00977 BC00977 VJ=100.00  +MOVJ EC00977 VJ=100.00
'Path S3472
SFTOF3D
MOVJ C00978 BC00978 VJ=100.00  +MOVJ EC00978 VJ=100.00
MOVL C00979 BC00979 V=666.7  +MOVJ EC00979 VJ=100.00
SMOVL C00980 BC00980 V=166.7  +MOVJ EC00980
SREFP 3 C00981 BC00981  +REFP EC00981
CALL JOB:SEARCH-R1-S13D
SET P032 P006
SFTON3D P032
SMOVL C00982 BC00982 V=166.7  +MOVJ EC00982
SREFP 3 C00983 BC00983  +REFP EC00983
CALL JOB:SEARCH-R1-S13D
SET P032 P006
SFTON3D P032
SMOVL C00984 BC00984 V=166.7  +MOVJ EC00984
SMOVL C00985 BC00985 V=133.3  +MOVJ EC00985
SREFP 3 C00986 BC00986  +REFP EC00986
CALL JOB:SEARCH-R1-S13D
SET P032 P006
SFTON3D P032
SMOVL C00987 BC00987 V=166.7  +MOVJ EC00987
MOVL C00988 BC00988 V=1000.0  +MOVJ EC00988 VJ=100.00
'EndPath S3472
MOVJ C00989 BC00989 VJ=100.00  +MOVJ EC00989 VJ=100.00
'Path S3477
SFTOF3D
MOVJ C00990 BC00990 VJ=100.00  +MOVJ EC00990 VJ=100.00
SMOVL C00991 BC00991 V=166.7  +MOVJ EC00991
SREFP 3 C00992 BC00992  +REFP EC00992
CALL JOB:SEARCH-R1-S13D
SET P069 P006
SFTON3D P069
SMOVL C00993 BC00993 V=250.0  +MOVJ EC00993
SMOVL C00994 BC00994 V=250.0  +MOVJ EC00994
SMOVL C00995 BC00995 V=166.7  +MOVJ EC00995
SREFP 3 C00996 BC00996  +REFP EC00996
CALL JOB:SEARCH-R1-S13D
SET P069 P006
SFTON3D P069
SMOVL C00997 BC00997 V=166.7  +MOVJ EC00997
SFTOF3D
SMOVL C00998 BC00998 V=666.7  +MOVJ EC00998
MOVL C00999 BC00999 V=666.7  +MOVJ EC00999 VJ=100.00
SMOVL C01000 BC01000 V=166.7  +MOVJ EC01000
SREFP 3 C01001 BC01001  +REFP EC01001
CALL JOB:SEARCH-R1-S13D
SET P052 P006
SFTON3D P052
SMOVL C01002 BC01002 V=166.7  +MOVJ EC01002
SREFP 3 C01003 BC01003  +REFP EC01003
CALL JOB:SEARCH-R1-S13D
SET P052 P006
SFTON3D P052
SMOVL C01004 BC01004 V=166.7  +MOVJ EC01004
MOVL C01005 BC01005 V=1000.0  +MOVJ EC01005 VJ=100.00
'EndPath S3477
MOVJ C01006 BC01006 VJ=100.00  +MOVJ EC01006 VJ=100.00
'poprawiÃÂ searcha- nie mialem
'wyciecia
'Path S3478
SFTOF3D
MOVJ C01007 BC01007 VJ=100.00  +MOVJ EC01007 VJ=100.00
MOVL C01008 BC01008 V=666.7  +MOVJ EC01008 VJ=100.00
SMOVL C01009 BC01009 V=166.7  +MOVJ EC01009
SREFP 3 C01010 BC01010  +REFP EC01010
CALL JOB:SEARCH-R1-S13D
SET P053 P006
SFTON3D P053
SMOVL C01011 BC01011 V=166.7  +MOVJ EC01011
SREFP 3 C01012 BC01012  +REFP EC01012
CALL JOB:SEARCH-R1-S13D
SET P053 P006
SFTON3D P053
SMOVL C01013 BC01013 V=166.7  +MOVJ EC01013
MOVL C01014 BC01014 V=1000.0  +MOVJ EC01014 VJ=100.00
'EndPath S3478
'
MOVJ C01015 BC01015 VJ=100.00  +MOVJ EC01015 VJ=100.00
'Path W3476
SFTOF3D
SFTON3D P033
MOVJ C01016 BC01016 VJ=100.00  +MOVJ EC01016 VJ=100.00
SMOVL C01017 BC01017 V=800.0  +MOVJ EC01017
SMOVL C01018 BC01018 V=166.7 PL=0  +MOVJ EC01018
MACRO1 MJ#(0) ARGF14
ARCON
SMOVL C01019 BC01019 V=10.0  +MOVJ EC01019
ARCOF
SMOVL C01020 BC01020 V=800.0  +MOVJ EC01020
SMOVL C01021 BC01021 V=1000.0  +MOVJ EC01021
SFTOF3D
'EndPath W3476
'Path W3477
SFTOF3D
SFTON3D P033
MOVJ C01022 BC01022 VJ=100.00  +MOVJ EC01022 VJ=100.00
SMOVL C01023 BC01023 V=800.0  +MOVJ EC01023
SMOVL C01024 BC01024 V=166.7 PL=0  +MOVJ EC01024
SMOVL C01025 BC01025 V=10.0  +MOVJ EC01025
SMOVL C01026 BC01026 V=10.0  +MOVJ EC01026
SMOVL C01027 BC01027 V=10.0  +MOVJ EC01027
ARCOF
SMOVL C01028 BC01028 V=800.0  +MOVJ EC01028
SMOVL C01029 BC01029 V=1000.0  +MOVJ EC01029
SFTOF3D
'EndPath W3477
MOVJ C01030 BC01030 VJ=100.00  +MOVJ EC01030 VJ=100.00
'Path W3478
SFTOF3D
SFTON3D P033
MOVJ C01031 BC01031 VJ=100.00  +MOVJ EC01031 VJ=100.00
SMOVL C01032 BC01032 V=800.0  +MOVJ EC01032
SMOVL C01033 BC01033 V=166.7 PL=0  +MOVJ EC01033
ARCON
SMOVL C01034 BC01034 V=10.0  +MOVJ EC01034
SMOVL C01035 BC01035 V=10.0  +MOVJ EC01035
SMOVL C01036 BC01036 V=10.0  +MOVJ EC01036
ARCOF
SMOVL C01037 BC01037 V=800.0  +MOVJ EC01037
SMOVL C01038 BC01038 V=1000.0  +MOVJ EC01038
SFTOF3D
'EndPath W3478
MOVJ C01039 BC01039 VJ=100.00  +MOVJ EC01039 VJ=100.00
MOVJ C01040 BC01040 VJ=100.00  +MOVJ EC01040 VJ=100.00
SFTOF3D
SFTON3D P081
MOVJ C01041 BC01041 VJ=100.00  +MOVJ EC01041 VJ=100.00
SMOVL C01042 BC01042 V=800.0  +MOVJ EC01042
SMOVL C01043 BC01043 V=166.7 PL=0  +MOVJ EC01043
ARCON
SMOVL C01044 BC01044 V=9.2  +MOVJ EC01044
ARCOF
SMOVL C01045 BC01045 V=800.0  +MOVJ EC01045
SMOVL C01046 BC01046 V=1000.0  +MOVJ EC01046
SFTOF3D
'EndPath W3479
'Path W3480
SFTOF3D
SFTON3D P081
MOVJ C01047 BC01047 VJ=100.00  +MOVJ EC01047 VJ=100.00
SMOVL C01048 BC01048 V=800.0  +MOVJ EC01048
SMOVL C01049 BC01049 V=150.0 PL=0  +MOVJ EC01049
ARCON
SMOVL C01050 BC01050 V=10.0  +MOVJ EC01050
ARCOF
SMOVL C01051 BC01051 V=800.0  +MOVJ EC01051
SMOVL C01052 BC01052 V=1000.0  +MOVJ EC01052
SFTOF3D
'EndPath W3480
'Path W3481
SFTOF3D
SFTON3D P081
MOVJ C01053 BC01053 VJ=100.00  +MOVJ EC01053 VJ=100.00
SMOVL C01054 BC01054 V=800.0  +MOVJ EC01054
SMOVL C01055 BC01055 V=150.0 PL=0  +MOVJ EC01055
ARCON
SMOVL C01056 BC01056 V=10.0  +MOVJ EC01056
ARCOF
SMOVL C01057 BC01057 V=800.0  +MOVJ EC01057
SMOVL C01058 BC01058 V=1000.0  +MOVJ EC01058
SFTOF3D
'EndPath W3481
MOVJ C01059 BC01059 VJ=100.00  +MOVJ EC01059 VJ=100.00
'uwaga na podajnik
'Path W3481
SFTOF3D
SFTON3D P081
MOVJ C01060 BC01060 VJ=50.00  +MOVJ EC01060 VJ=15.00
SMOVL C01061 BC01061 V=800.0  +MOVJ EC01061
SMOVL C01062 BC01062 V=150.0 PL=0  +MOVJ EC01062
ARCON
SMOVL C01063 BC01063 V=10.0  +MOVJ EC01063
ARCOF
SMOVL C01064 BC01064 V=800.0  +MOVJ EC01064
SMOVL C01065 BC01065 V=1000.0  +MOVJ EC01065
SFTOF3D
'9
'Path W3479
MOVJ C01066 BC01066 VJ=100.00  +MOVJ EC01066 VJ=100.00
SFTOF3D
SFTON3D P026
MOVJ C01067 BC01067 VJ=100.00  +MOVJ EC01067 VJ=100.00
SMOVL C01068 BC01068 V=800.0  +MOVJ EC01068
SMOVL C01069 BC01069 V=166.7 PL=0  +MOVJ EC01069
ARCON
SMOVL C01070 BC01070 V=9.2  +MOVJ EC01070
SMOVL C01071 BC01071 V=9.2  +MOVJ EC01071
SMOVL C01072 BC01072 V=9.2  +MOVJ EC01072
ARCOF
SMOVL C01073 BC01073 V=800.0  +MOVJ EC01073
SMOVL C01074 BC01074 V=1000.0  +MOVJ EC01074
SFTOF3D
'EndPath W3479
'Path W3480
SFTOF3D
SFTON3D P026
MOVJ C01075 BC01075 VJ=100.00  +MOVJ EC01075 VJ=100.00
SMOVL C01076 BC01076 V=800.0  +MOVJ EC01076
SMOVL C01077 BC01077 V=150.0 PL=0  +MOVJ EC01077
ARCON
SMOVL C01078 BC01078 V=10.0  +MOVJ EC01078
SMOVL C01079 BC01079 V=10.0  +MOVJ EC01079
SMOVL C01080 BC01080 V=10.0  +MOVJ EC01080
ARCOF
SMOVL C01081 BC01081 V=800.0  +MOVJ EC01081
SMOVL C01082 BC01082 V=1000.0  +MOVJ EC01082
SFTOF3D
'EndPath W3480
'Path W3481
SFTOF3D
SFTON3D P026
MOVJ C01083 BC01083 VJ=100.00  +MOVJ EC01083 VJ=100.00
SMOVL C01084 BC01084 V=800.0  +MOVJ EC01084
SMOVL C01085 BC01085 V=150.0 PL=0  +MOVJ EC01085
ARCON
SMOVL C01086 BC01086 V=10.0  +MOVJ EC01086
ARCOF
SMOVL C01087 BC01087 V=800.0  +MOVJ EC01087
SMOVL C01088 BC01088 V=1000.0  +MOVJ EC01088
SFTOF3D
'EndPath W3481
MOVJ C01089 BC01089 VJ=100.00  +MOVJ EC01089 VJ=100.00
'uwaga na podajnik
'Path W3481
SFTOF3D
SFTON3D P026
MOVJ C01090 BC01090 VJ=50.00  +MOVJ EC01090 VJ=15.00
SMOVL C01091 BC01091 V=800.0  +MOVJ EC01091
SMOVL C01092 BC01092 V=150.0 PL=0  +MOVJ EC01092
ARCON
SMOVL C01093 BC01093 V=10.0  +MOVJ EC01093
SMOVL C01094 BC01094 V=10.0  +MOVJ EC01094
ARCOF
SMOVL C01095 BC01095 V=800.0  +MOVJ EC01095
SMOVL C01096 BC01096 V=1000.0  +MOVJ EC01096
SFTOF3D
'EndPath W3481
'brak dostepu offset drutu 1cm
'Path W3482
SFTOF3D
SFTON3D P026
MOVJ C01097 BC01097 VJ=100.00  +MOVJ EC01097 VJ=100.00
SMOVL C01098 BC01098 V=800.0  +MOVJ EC01098
SMOVL C01099 BC01099 V=150.0 PL=0  +MOVJ EC01099
ARCON
SMOVL C01100 BC01100 V=10.0  +MOVJ EC01100
ARCOF
SMOVL C01101 BC01101 V=800.0  +MOVJ EC01101
SMOVL C01102 BC01102 V=1000.0  +MOVJ EC01102
SFTOF3D
'EndPath W3482
MOVJ C01103 BC01103 VJ=100.00  +MOVJ EC01103 VJ=100.00
MOVJ C01104 BC01104 VJ=100.00  +MOVJ EC01104 VJ=100.00
'10
'11
'Path W3484
SFTOF3D
SFTON3D P025
MOVJ C01105 BC01105 VJ=100.00  +MOVJ EC01105 VJ=100.00
SMOVL C01106 BC01106 V=800.0  +MOVJ EC01106
SMOVL C01107 BC01107 V=150.0 PL=0  +MOVJ EC01107
ARCON
SMOVL C01108 BC01108 V=10.0  +MOVJ EC01108
SMOVL C01109 BC01109 V=10.0  +MOVJ EC01109
ARCOF
SMOVL C01110 BC01110 V=800.0  +MOVJ EC01110
SMOVL C01111 BC01111 V=1000.0  +MOVJ EC01111
SFTOF3D
'EndPath W3484
MOVJ C01112 BC01112 VJ=100.00  +MOVJ EC01112 VJ=100.00
'brak dostepu offset drutu 1cm
'Path W3483
SFTOF3D
SFTON3D P025
MOVJ C01113 BC01113 VJ=100.00  +MOVJ EC01113 VJ=100.00
SMOVL C01114 BC01114 V=800.0  +MOVJ EC01114
SMOVL C01115 BC01115 V=166.7 PL=0  +MOVJ EC01115
ARCON
SMOVL C01116 BC01116 V=10.0  +MOVJ EC01116
ARCOF
SMOVL C01117 BC01117 V=800.0  +MOVJ EC01117
SMOVL C01118 BC01118 V=1000.0  +MOVJ EC01118
SFTOF3D
'EndPath W3483
MOVJ C01119 BC01119 VJ=100.00  +MOVJ EC01119 VJ=100.00
MOVJ C01120 BC01120 VJ=100.00  +MOVJ EC01120 VJ=100.00
MOVJ C01121 BC01121 VJ=100.00  +MOVJ EC01121 VJ=100.00
'Path W4854
SFTOF3D
SFTON3D P073
MOVJ C01122 BC01122 VJ=100.00  +MOVJ EC01122 VJ=100.00
SMOVL C01123 BC01123 V=800.0  +MOVJ EC01123
SMOVL C01124 BC01124 V=150.0 PL=0  +MOVJ EC01124
MACRO1 MJ#(0) ARGF9
ARCON
SMOVL C01125 BC01125 V=9.2  +MOVJ EC01125
SFTON3D P074
SMOVL C01126 BC01126 V=9.2  +MOVJ EC01126
SMOVL C01127 BC01127 V=9.2  +MOVJ EC01127
ARCOF
SMOVL C01128 BC01128 V=800.0  +MOVJ EC01128
MOVJ C01129 BC01129 VJ=50.00  +MOVJ EC01129 VJ=100.00
SMOVL C01130 BC01130 V=166.7  +MOVJ EC01130
SMOVL C01131 BC01131 V=166.7  +MOVJ EC01131
SMOVL C01132 BC01132 V=50.0 PL=0  +MOVJ EC01132
ARCON
SMOVL C01133 BC01133 V=9.2  +MOVJ EC01133
SMOVL C01134 BC01134 V=9.2  +MOVJ EC01134
ARCOF
SMOVL C01135 BC01135 V=1000.0  +MOVJ EC01135
SFTOF3D
'EndPath W4854
'12
MOVJ C01136 BC01136 VJ=100.00  +MOVJ EC01136 VJ=100.00
MOVJ C01137 BC01137 VJ=100.00  +MOVJ EC01137 VJ=100.00
MOVJ C01138 BC01138 VJ=100.00  +MOVJ EC01138 VJ=100.00
'Path W3485
SFTOF3D
SFTON3D P034
MOVJ C01139 BC01139 VJ=100.00  +MOVJ EC01139 VJ=100.00
SMOVL C01140 BC01140 V=800.0  +MOVJ EC01140
SMOVL C01141 BC01141 V=150.0 PL=0  +MOVJ EC01141
MACRO1 MJ#(0) ARGF14
ARCON
SMOVL C01142 BC01142 V=10.0  +MOVJ EC01142
SMOVL C01143 BC01143 V=10.0  +MOVJ EC01143
SMOVL C01144 BC01144 V=10.0  +MOVJ EC01144
ARCOF
SMOVL C01145 BC01145 V=800.0  +MOVJ EC01145
SMOVL C01146 BC01146 V=1000.0  +MOVJ EC01146
SFTOF3D
MOVJ C01147 BC01147 VJ=80.00  +MOVJ EC01147 VJ=80.00
MOVJ C01148 BC01148 VJ=80.00  +MOVJ EC01148 VJ=80.00
MOVJ C01149 BC01149 VJ=80.00  +MOVJ EC01149 VJ=80.00
MACRO1 MJ#(0) ARGF6
SFTON3D P063
SMOVL C01150 BC01150 V=166.7  +MOVJ EC01150
ARCON
SMOVL C01151 BC01151 V=11.7  +MOVJ EC01151
SMOVL C01152 BC01152 V=11.7  +MOVJ EC01152
SFTON3D P062
SMOVL C01153 BC01153 V=11.0  +MOVJ EC01153
SMOVL C01154 BC01154 V=11.0  +MOVJ EC01154
SFTON3D P061
SMOVL C01155 BC01155 V=11.0  +MOVJ EC01155
SMOVL C01156 BC01156 V=11.0  +MOVJ EC01156
ARCOF
SMOVL C01157 BC01157 V=800.0  +MOVJ EC01157
SFTOF3D
MOVJ C01158 BC01158 VJ=80.00  +MOVJ EC01158 VJ=80.00
MOVJ C01159 BC01159 VJ=80.00  +MOVJ EC01159 VJ=80.00
MOVJ C01160 BC01160 VJ=80.00  +MOVJ EC01160 VJ=80.00
'EndPath W3485
'Path W3486
SFTOF3D
SFTON3D P050
MOVJ C01161 BC01161 VJ=100.00  +MOVJ EC01161 VJ=100.00
SMOVL C01162 BC01162 V=800.0  +MOVJ EC01162
SMOVL C01163 BC01163 V=150.0 PL=0  +MOVJ EC01163
MACRO1 MJ#(0) ARGF14
ARCON
SMOVL C01164 BC01164 V=10.0  +MOVJ EC01164
SMOVL C01165 BC01165 V=10.0  +MOVJ EC01165
SMOVL C01166 BC01166 V=10.0  +MOVJ EC01166
ARCOF
SMOVL C01167 BC01167 V=800.0  +MOVJ EC01167
SMOVL C01168 BC01168 V=1000.0  +MOVJ EC01168
SFTOF3D
'EndPath W3486
MOVJ C01169 BC01169 VJ=100.00  +MOVJ EC01169 VJ=100.00
'Path W3485
SFTOF3D
SFTON3D P034
MOVJ C01170 BC01170 VJ=100.00  +MOVJ EC01170 VJ=100.00
SMOVL C01171 BC01171 V=800.0  +MOVJ EC01171
SMOVL C01172 BC01172 V=166.7 PL=0  +MOVJ EC01172
SREFP 1 C01173 BC01173  +REFP EC01173
SREFP 2 C01174 BC01174  +REFP EC01174
ARCON
SWVON WEV#(20)
SMOVL C01175 BC01175 V=9.2  +MOVJ EC01175
SMOVL C01176 BC01176 V=9.2  +MOVJ EC01176
SMOVL C01177 BC01177 V=9.2  +MOVJ EC01177
ARCOF
SWVOF
SMOVL C01178 BC01178 V=800.0  +MOVJ EC01178
SMOVL C01179 BC01179 V=1000.0  +MOVJ EC01179
SFTOF3D
'EndPath W3485
'Path W3487
SFTOF3D
SFTON3D P054
MOVJ C01180 BC01180 VJ=100.00  +MOVJ EC01180 VJ=100.00
SMOVL C01181 BC01181 V=800.0  +MOVJ EC01181
SMOVL C01182 BC01182 V=150.0 PL=0  +MOVJ EC01182
ARCON
SWVON WEV#(20)
SMOVL C01183 BC01183 V=9.2  +MOVJ EC01183
SMOVL C01184 BC01184 V=9.2  +MOVJ EC01184
SMOVL C01185 BC01185 V=9.2  +MOVJ EC01185
ARCOF
SWVOF
SMOVL C01186 BC01186 V=800.0  +MOVJ EC01186
SMOVL C01187 BC01187 V=1000.0  +MOVJ EC01187
SFTOF3D
'EndPath W3487
MOVJ C01188 BC01188 VJ=100.00  +MOVJ EC01188 VJ=100.00
'Path W3487
SFTOF3D
SFTON3D P028
MOVJ C01189 BC01189 VJ=100.00  +MOVJ EC01189 VJ=100.00
SMOVL C01190 BC01190 V=800.0  +MOVJ EC01190
SMOVL C01191 BC01191 V=150.0 PL=0  +MOVJ EC01191
ARCON
SMOVL C01192 BC01192 V=9.2  +MOVJ EC01192
SMOVL C01193 BC01193 V=9.2  +MOVJ EC01193
SMOVL C01194 BC01194 V=9.2  +MOVJ EC01194
ARCOF
SMOVL C01195 BC01195 V=800.0  +MOVJ EC01195
SMOVL C01196 BC01196 V=1000.0  +MOVJ EC01196
SFTOF3D
'EndPath W3487
MOVJ C01197 BC01197 VJ=100.00  +MOVJ EC01197 VJ=100.00
MOVJ C01198 BC01198 VJ=100.00  +MOVJ EC01198 VJ=100.00
'brak dostepu offset 5mm
'Path W3488
SFTOF3D
SFTON3D P028
MOVJ C01199 BC01199 VJ=100.00  +MOVJ EC01199 VJ=100.00
SMOVL C01200 BC01200 V=800.0  +MOVJ EC01200
SMOVL C01201 BC01201 V=150.0 PL=0  +MOVJ EC01201
ARCON
SMOVL C01202 BC01202 V=11.7  +MOVJ EC01202
ARCOF
SMOVL C01203 BC01203 V=800.0  +MOVJ EC01203
SMOVL C01204 BC01204 V=1000.0  +MOVJ EC01204
SFTOF3D
'EndPath W3488
MOVJ C01205 BC01205 VJ=100.00  +MOVJ EC01205 VJ=100.00
'13
'Path W3489
SFTOF3D
SFTON3D P030
MOVJ C01206 BC01206 VJ=100.00  +MOVJ EC01206 VJ=100.00
SMOVL C01207 BC01207 V=800.0  +MOVJ EC01207
SMOVL C01208 BC01208 V=150.0 PL=0  +MOVJ EC01208
MACRO1 MJ#(0) ARGF9
ARCON
SWVON WEV#(10)
SFTON3D P031
SMOVL C01209 BC01209 V=12.5  +MOVJ EC01209
SFTON3D P098
SMOVL C01210 BC01210 V=12.5  +MOVJ EC01210
ARCOF
SWVOF
SMOVL C01211 BC01211 V=800.0  +MOVJ EC01211
SMOVL C01212 BC01212 V=1000.0  +MOVJ EC01212
SFTOF3D
'EndPath W3489
'Path W3490
SFTOF3D
MOVJ C01213 BC01213 VJ=100.00  +MOVJ EC01213 VJ=100.00
MACRO1 MJ#(0) ARGF6
SFTON3D P069
SMOVL C01214 BC01214 V=250.0  +MOVJ EC01214
ARCON
SMOVL C01215 BC01215 V=11.7  +MOVJ EC01215
ARCOF
SMOVL C01216 BC01216 V=250.0  +MOVJ EC01216
SFTOF3D
SFTON3D P052
MOVJ C01217 BC01217 VJ=100.00  +MOVJ EC01217 VJ=100.00
SMOVL C01218 BC01218 V=800.0  +MOVJ EC01218
SMOVL C01219 BC01219 V=150.0 PL=0  +MOVJ EC01219
MACRO1 MJ#(0) ARGF14
ARCON
SMOVL C01220 BC01220 V=10.0  +MOVJ EC01220
SMOVL C01221 BC01221 V=10.0  +MOVJ EC01221
SMOVL C01222 BC01222 V=10.0  +MOVJ EC01222
ARCOF
SMOVL C01223 BC01223 V=800.0  +MOVJ EC01223
SMOVL C01224 BC01224 V=1000.0  +MOVJ EC01224
SFTOF3D
'EndPath W3490
MOVJ C01225 BC01225 VJ=100.00  +MOVJ EC01225 VJ=100.00
'poprawic spoine - nie mialem w
'yciecia
'Path W3491
SFTOF3D
SFTON3D P053
MOVJ C01226 BC01226 VJ=100.00  +MOVJ EC01226 VJ=100.00
SMOVL C01227 BC01227 V=800.0  +MOVJ EC01227
SMOVL C01228 BC01228 V=150.0 PL=0  +MOVJ EC01228
ARCON
SMOVL C01229 BC01229 V=10.0  +MOVJ EC01229
SMOVL C01230 BC01230 V=10.0  +MOVJ EC01230
SMOVL C01231 BC01231 V=10.0  +MOVJ EC01231
ARCOF
SMOVL C01232 BC01232 V=800.0  +MOVJ EC01232
SMOVL C01233 BC01233 V=1000.0  +MOVJ EC01233
SFTOF3D
'EndPath W3491
'14
'15-brak
MOVJ C01234 BC01234 VJ=100.00  +MOVJ EC01234 VJ=100.00
'16
'Path W3491
SFTOF3D
SFTON3D P029
MOVJ C01235 BC01235 VJ=100.00  +MOVJ EC01235 VJ=100.00
SMOVL C01236 BC01236 V=800.0  +MOVJ EC01236
SMOVL C01237 BC01237 V=150.0 PL=0  +MOVJ EC01237
COMM ARCON
SMOVL C01238 BC01238 V=10.0  +MOVJ EC01238
SMOVL C01239 BC01239 V=10.0  +MOVJ EC01239
ARCOF
SMOVL C01240 BC01240 V=800.0  +MOVJ EC01240
SMOVL C01241 BC01241 V=1000.0  +MOVJ EC01241
SFTOF3D
'EndPath W3491
MOVJ C01242 BC01242 VJ=100.00  +MOVJ EC01242 VJ=100.00
'Path W3492
SFTOF3D
SFTON3D P029
MOVJ C01243 BC01243 VJ=100.00  +MOVJ EC01243 VJ=100.00
SMOVL C01244 BC01244 V=800.0  +MOVJ EC01244
SMOVL C01245 BC01245 V=150.0 PL=0  +MOVJ EC01245
COMM ARCON
SMOVL C01246 BC01246 V=10.0  +MOVJ EC01246
ARCOF
SMOVL C01247 BC01247 V=800.0  +MOVJ EC01247
SMOVL C01248 BC01248 V=1000.0  +MOVJ EC01248
SFTOF3D
'EndPath W3492
MOVJ C01249 BC01249 VJ=100.00  +MOVJ EC01249 VJ=100.00
MOVJ C01250 BC01250 VJ=100.00  +MOVJ EC01250 VJ=100.00
'Path W3493
SFTOF3D
SFTON3D P029
MOVJ C01251 BC01251 VJ=100.00  +MOVJ EC01251 VJ=100.00
SMOVL C01252 BC01252 V=800.0  +MOVJ EC01252
SMOVL C01253 BC01253 V=150.0 PL=0  +MOVJ EC01253
COMM ARCON
SMOVL C01254 BC01254 V=10.0  +MOVJ EC01254
SMOVL C01255 BC01255 V=10.0  +MOVJ EC01255
SMOVL C01256 BC01256 V=10.0  +MOVJ EC01256
ARCON
SMOVL C01257 BC01257 V=11.7  +MOVJ EC01257
ARCON
SMOVL C01258 BC01258 V=11.7  +MOVJ EC01258
ARCOF
SMOVL C01259 BC01259 V=800.0  +MOVJ EC01259
SMOVL C01260 BC01260 V=1000.0  +MOVJ EC01260
SFTOF3D
'EndPath W3493
MOVJ C01261 BC01261 VJ=100.00  +MOVJ EC01261 VJ=100.00
MOVJ C01262 BC01262 VJ=100.00  +MOVJ EC01262 VJ=100.00
'16
'Path W3491
SFTOF3D
SFTON3D P080
MOVJ C01263 BC01263 VJ=100.00  +MOVJ EC01263 VJ=100.00
SMOVL C01264 BC01264 V=800.0  +MOVJ EC01264
SMOVL C01265 BC01265 V=150.0 PL=0  +MOVJ EC01265
ARCON
SMOVL C01266 BC01266 V=10.0  +MOVJ EC01266
SMOVL C01267 BC01267 V=10.0  +MOVJ EC01267
ARCOF
SMOVL C01268 BC01268 V=800.0  +MOVJ EC01268
SMOVL C01269 BC01269 V=1000.0  +MOVJ EC01269
SFTOF3D
'EndPath W3491
MOVJ C01270 BC01270 VJ=100.00  +MOVJ EC01270 VJ=100.00
'Path W3492
SFTOF3D
SFTON3D P080
MOVJ C01271 BC01271 VJ=100.00  +MOVJ EC01271 VJ=100.00
SMOVL C01272 BC01272 V=800.0  +MOVJ EC01272
SMOVL C01273 BC01273 V=150.0 PL=0  +MOVJ EC01273
ARCON
SMOVL C01274 BC01274 V=10.0  +MOVJ EC01274
ARCOF
SMOVL C01275 BC01275 V=800.0  +MOVJ EC01275
SMOVL C01276 BC01276 V=1000.0  +MOVJ EC01276
SFTOF3D
'EndPath W3492
MOVJ C01277 BC01277 VJ=100.00  +MOVJ EC01277 VJ=100.00
MOVJ C01278 BC01278 VJ=100.00  +MOVJ EC01278 VJ=100.00
'Path W3493
SFTOF3D
SFTON3D P080
MOVJ C01279 BC01279 VJ=100.00  +MOVJ EC01279 VJ=100.00
SMOVL C01280 BC01280 V=800.0  +MOVJ EC01280
SMOVL C01281 BC01281 V=150.0 PL=0  +MOVJ EC01281
ARCON
SMOVL C01282 BC01282 V=10.0  +MOVJ EC01282
SMOVL C01283 BC01283 V=10.0  +MOVJ EC01283
SMOVL C01284 BC01284 V=10.0  +MOVJ EC01284
ARCON
SMOVL C01285 BC01285 V=11.7  +MOVJ EC01285
ARCON
SMOVL C01286 BC01286 V=11.7  +MOVJ EC01286
ARCOF
SMOVL C01287 BC01287 V=800.0  +MOVJ EC01287
SMOVL C01288 BC01288 V=1000.0  +MOVJ EC01288
SFTOF3D
'EndPath W3493
MOVJ C01289 BC01289 VJ=100.00  +MOVJ EC01289 VJ=100.00
MOVJ C01290 BC01290 VJ=100.00  +MOVJ EC01290 VJ=100.00
'17
'Path W3494
SFTOF3D
SFTON3D P027
MOVJ C01291 BC01291 VJ=100.00  +MOVJ EC01291 VJ=100.00
SMOVL C01292 BC01292 V=800.0  +MOVJ EC01292
SMOVL C01293 BC01293 V=150.0 PL=0  +MOVJ EC01293
ARCON
SMOVL C01294 BC01294 V=10.0  +MOVJ EC01294
ARCOF
SMOVL C01295 BC01295 V=800.0  +MOVJ EC01295
SMOVL C01296 BC01296 V=1000.0  +MOVJ EC01296
SFTOF3D
'EndPath W3494
'Path W3495
SFTOF3D
SFTON3D P027
MOVJ C01297 BC01297 VJ=100.00  +MOVJ EC01297 VJ=100.00
SMOVL C01298 BC01298 V=800.0  +MOVJ EC01298
SMOVL C01299 BC01299 V=150.0 PL=0  +MOVJ EC01299
ARCON
SMOVL C01300 BC01300 V=10.8  +MOVJ EC01300
ARCOF
SMOVL C01301 BC01301 V=800.0  +MOVJ EC01301
SMOVL C01302 BC01302 V=1000.0  +MOVJ EC01302
SFTOF3D
'EndPath W3495
'Path W3496
SFTOF3D
SFTON3D P027
MOVJ C01303 BC01303 VJ=100.00  +MOVJ EC01303 VJ=100.00
SFTOF3D
'EndPath W3496
MOVJ C01304 BC01304 VJ=100.00  +MOVJ EC01304 VJ=100.00
MOVJ C01305 BC01305 VJ=100.00  +MOVJ EC01305 VJ=100.00
MOVJ C01306 BC01306 VJ=100.00  +MOVJ EC01306 VJ=100.00
'18
'Path W3497
SFTOF3D
SFTON3D P024
MOVJ C01307 BC01307 VJ=100.00  +MOVJ EC01307 VJ=100.00
SMOVL C01308 BC01308 V=800.0  +MOVJ EC01308
SMOVL C01309 BC01309 V=150.0 PL=0  +MOVJ EC01309
COMM ARCON
SMOVL C01310 BC01310 V=9.2  +MOVJ EC01310
SMOVL C01311 BC01311 V=9.2  +MOVJ EC01311
SMOVL C01312 BC01312 V=9.2  +MOVJ EC01312
SMOVL C01313 BC01313 V=9.2  +MOVJ EC01313
ARCOF
SMOVL C01314 BC01314 V=800.0  +MOVJ EC01314
SMOVL C01315 BC01315 V=1000.0  +MOVJ EC01315
SFTOF3D
'EndPath W3497
'
'Path W4855
SFTOF3D
SFTON3D P071
MOVJ C01316 BC01316 VJ=100.00  +MOVJ EC01316 VJ=100.00
SMOVL C01317 BC01317 V=800.0  +MOVJ EC01317
MACRO1 MJ#(0) ARGF9
SMOVL C01318 BC01318 V=150.0 PL=0  +MOVJ EC01318
ARCON
SMOVL C01319 BC01319 V=8.8  +MOVJ EC01319
SFTON3D P072
SMOVL C01320 BC01320 V=8.8  +MOVJ EC01320
SMOVL C01321 BC01321 V=8.8  +MOVJ EC01321
ARCOF
SMOVL C01322 BC01322 V=166.7  +MOVJ EC01322
SMOVL C01323 BC01323 V=800.0  +MOVJ EC01323
SMOVL C01324 BC01324 V=800.0  +MOVJ EC01324
SMOVL C01325 BC01325 V=800.0  +MOVJ EC01325
SFTON3D P072
SMOVL C01326 BC01326 V=166.7 PL=0  +MOVJ EC01326
ARCON
SMOVL C01327 BC01327 V=8.8  +MOVJ EC01327
SMOVL C01328 BC01328 V=8.8  +MOVJ EC01328
SMOVL C01329 BC01329 V=8.8  +MOVJ EC01329
SMOVL C01330 BC01330 V=8.8  +MOVJ EC01330
ARCOF
MOVL C01331 BC01331 V=166.7  +MOVJ EC01331 VJ=0.78
SMOVL C01332 BC01332 V=1000.0  +MOVJ EC01332
SFTOF3D
'EndPath W4855
'
'
MOVJ C01333 BC01333 VJ=100.00  +MOVJ EC01333 VJ=100.00
'19
MOVJ C01334 BC01334 VJ=100.00  +MOVJ EC01334 VJ=100.00
'Path W3499
SFTOF3D
SFTON3D P023
MOVJ C01335 BC01335 VJ=100.00  +MOVJ EC01335 VJ=100.00
SMOVL C01336 BC01336 V=800.0  +MOVJ EC01336
SMOVL C01337 BC01337 V=150.0 PL=0  +MOVJ EC01337
MACRO1 MJ#(0) ARGF6
ARCON
SWVON WEV#(66)
SMOVL C01338 BC01338 V=7.5  +MOVJ EC01338
SMOVL C01339 BC01339 V=7.5  +MOVJ EC01339
SMOVL C01340 BC01340 V=7.5  +MOVJ EC01340
ARCOF
SWVOF
SMOVL C01341 BC01341 V=800.0  +MOVJ EC01341
SMOVL C01342 BC01342 V=1000.0  +MOVJ EC01342
SFTOF3D
'EndPath W3499
MOVJ C01343 BC01343 VJ=100.00  +MOVJ EC01343 VJ=100.00
'Path W3500
SFTOF3D
SFTON3D P034
MOVJ C01344 BC01344 VJ=100.00  +MOVJ EC01344 VJ=100.00
SMOVL C01345 BC01345 V=800.0  +MOVJ EC01345
MACRO1 MJ#(0) ARGF9
SMOVL C01346 BC01346 V=150.0 PL=0  +MOVJ EC01346
ARCON
SMOVL C01347 BC01347 V=8.3  +MOVJ EC01347
SFTON3D P050
SMOVL C01348 BC01348 V=8.3  +MOVJ EC01348
SMOVL C01349 BC01349 V=8.3  +MOVJ EC01349
ARCOF
SMOVL C01350 BC01350 V=800.0  +MOVJ EC01350
SMOVL C01351 BC01351 V=1000.0  +MOVJ EC01351
SFTOF3D
'EndPath W3500
'Path W3501
SFTOF3D
SFTON3D P051
MOVJ C01352 BC01352 VJ=100.00  +MOVJ EC01352 VJ=100.00
SMOVL C01353 BC01353 V=800.0  +MOVJ EC01353
SMOVL C01354 BC01354 V=150.0 PL=0  +MOVJ EC01354
ARCON
SWVON WEV#(60)
SMOVL C01355 BC01355 V=7.5  +MOVJ EC01355
SMOVL C01356 BC01356 V=7.5  +MOVJ EC01356
SMOVL C01357 BC01357 V=7.5  +MOVJ EC01357
ARCOF
SWVOF
SMOVL C01358 BC01358 V=800.0  +MOVJ EC01358
SMOVL C01359 BC01359 V=1000.0  +MOVJ EC01359
SFTOF3D
'EndPath W3501
MOVJ C01360 BC01360 VJ=100.00  +MOVJ EC01360 VJ=100.00
'20
MOVJ C01361 BC01361 VJ=100.00  +MOVJ EC01361 VJ=100.00
MOVJ C01362 BC01362 VJ=100.00  +MOVJ EC01362 VJ=100.00
'offset 5mm
'Path W3500
SFTOF3D
SFTON3D P032
MOVJ C01363 BC01363 VJ=100.00  +MOVJ EC01363 VJ=100.00
SMOVL C01364 BC01364 V=800.0  +MOVJ EC01364
SMOVL C01365 BC01365 V=150.0 PL=0  +MOVJ EC01365
ARCON
SMOVL C01366 BC01366 V=9.2  +MOVJ EC01366
ARCOF
SMOVL C01367 BC01367 V=800.0  +MOVJ EC01367
SMOVL C01368 BC01368 V=1000.0  +MOVJ EC01368
SFTOF3D
'EndPath W3500
SFTOF3D
'EndPath W3502
'offset 5mm
'Path W3503
SFTOF3D
SFTON3D P032
MOVJ C01369 BC01369 VJ=100.00  +MOVJ EC01369 VJ=100.00
SMOVL C01370 BC01370 V=800.0  +MOVJ EC01370
SMOVL C01371 BC01371 V=150.0 PL=0  +MOVJ EC01371
ARCON
SMOVL C01372 BC01372 V=10.0  +MOVJ EC01372
ARCOF
SMOVL C01373 BC01373 V=800.0  +MOVJ EC01373
SMOVL C01374 BC01374 V=1000.0  +MOVJ EC01374
SFTOF3D
'EndPath W3503
MOVJ C01375 BC01375 VJ=100.00  +MOVJ EC01375 VJ=100.00
'Path W3504
SFTOF3D
SFTON3D P032
MOVJ C01376 BC01376 VJ=100.00  +MOVJ EC01376 VJ=100.00
SMOVL C01377 BC01377 V=800.0  +MOVJ EC01377
SMOVL C01378 BC01378 V=150.0 PL=0  +MOVJ EC01378
ARCON
SMOVL C01379 BC01379 V=11.7  +MOVJ EC01379
SMOVL C01380 BC01380 V=11.7  +MOVJ EC01380
ARCOF
SMOVL C01381 BC01381 V=800.0  +MOVJ EC01381
SMOVL C01382 BC01382 V=1000.0  +MOVJ EC01382
SFTOF3D
'EndPath W3504
MOVJ C01383 BC01383 VJ=100.00  +MOVJ EC01383 VJ=100.00
'21
MOVJ C01384 BC01384 VJ=100.00  +MOVJ EC01384 VJ=100.00
'Path W3505
SFTOF3D
SFTON3D P097
MOVJ C01385 BC01385 VJ=100.00  +MOVJ EC01385 VJ=100.00
SMOVL C01386 BC01386 V=800.0  +MOVJ EC01386
SMOVL C01387 BC01387 V=150.0 PL=0  +MOVJ EC01387
ARCON
SMOVL C01388 BC01388 V=10.8  +MOVJ EC01388
SFTON3D P021
SMOVL C01389 BC01389 V=10.8  +MOVJ EC01389
SFTON3D P022
SMOVL C01390 BC01390 V=10.8  +MOVJ EC01390
SMOVL C01391 BC01391 V=11.7  +MOVJ EC01391
ARCOF
SMOVL C01392 BC01392 V=800.0  +MOVJ EC01392
SMOVL C01393 BC01393 V=1000.0  +MOVJ EC01393
SFTOF3D
'EndPath W3505
MOVJ C01394 BC01394 VJ=100.00  +MOVJ EC01394 VJ=100.00
'Path W3506
SFTOF3D
SFTON3D P095
MOVJ C01395 BC01395 VJ=100.00  +MOVJ EC01395 VJ=100.00
SMOVL C01396 BC01396 V=800.0  +MOVJ EC01396
SMOVL C01397 BC01397 V=150.0 PL=0  +MOVJ EC01397
MACRO1 MJ#(0) ARGF14
ARCON
SMOVL C01398 BC01398 V=10.0  +MOVJ EC01398
SMOVL C01399 BC01399 V=10.0  +MOVJ EC01399
SMOVL C01400 BC01400 V=10.0  +MOVJ EC01400
ARCOF
SMOVL C01401 BC01401 V=800.0  +MOVJ EC01401
SMOVL C01402 BC01402 V=1000.0  +MOVJ EC01402
SFTOF3D
'EndPath W3506
'Path W3507
SFTOF3D
SFTON3D P096
MOVJ C01403 BC01403 VJ=100.00  +MOVJ EC01403 VJ=100.00
SMOVL C01404 BC01404 V=800.0  +MOVJ EC01404
SMOVL C01405 BC01405 V=150.0 PL=0  +MOVJ EC01405
ARCON
SMOVL C01406 BC01406 V=10.0  +MOVJ EC01406
SMOVL C01407 BC01407 V=10.0  +MOVJ EC01407
ARCOF
SMOVL C01408 BC01408 V=800.0  +MOVJ EC01408
SMOVL C01409 BC01409 V=1000.0  +MOVJ EC01409
SFTOF3D
'EndPath W3507
MOVJ C01410 BC01410 VJ=100.00  +MOVJ EC01410 VJ=100.00
MOVJ C01411 BC01411 VJ=100.00  +MOVJ EC01411 VJ=100.00
'Path W4856
SFTOF3D
SFTON3D P071
MOVJ C01412 BC01412 VJ=100.00  +MOVJ EC01412 VJ=100.00
SMOVL C01413 BC01413 V=800.0  +MOVJ EC01413
SMOVL C01414 BC01414 V=150.0 PL=0  +MOVJ EC01414
ARCON
SMOVL C01415 BC01415 V=8.3  +MOVJ EC01415
SFTON3D P073
SMOVL C01416 BC01416 V=8.3  +MOVJ EC01416
SMOVL C01417 BC01417 V=8.3  +MOVJ EC01417
ARCOF
SMOVL C01418 BC01418 V=800.0  +MOVJ EC01418
SMOVL C01419 BC01419 V=1000.0  +MOVJ EC01419
SFTOF3D
'EndPath W4856
MOVJ C01420 BC01420 VJ=100.00  +MOVJ EC01420 VJ=100.00
MOVJ C01421 BC01421 VJ=50.00  +MOVJ EC01421 VJ=0.78
MOVJ C01422 BC01422 VJ=100.00  +MOVJ EC01422 VJ=50.00
SFTON3D P080
SMOVL C01423 BC01423 V=800.0  +MOVJ EC01423
SMOVL C01424 BC01424 V=150.0 PL=0  +MOVJ EC01424
ARCON
SMOVL C01425 BC01425 V=8.3  +MOVJ EC01425
SMOVL C01426 BC01426 V=8.3  +MOVJ EC01426
SMOVC C01427 BC01427 V=8.3  +MOVJ EC01427
ARCOF
SMOVL C01428 BC01428 V=800.0  +MOVJ EC01428
SFTOF3D
SMOVL C01429 BC01429 V=1000.0  +MOVJ EC01429
MOVJ C01430 BC01430 VJ=100.00  +MOVJ EC01430 VJ=100.00
MOVJ C01431 BC01431 VJ=100.00  +MOVJ EC01431 VJ=100.00
MOVJ C01432 BC01432 VJ=100.00  +MOVJ EC01432 VJ=100.00
MOVJ C01433 BC01433 VJ=100.00  +MOVJ EC01433 VJ=100.00
SFTON3D P081
SMOVL C01434 BC01434 V=666.7  +MOVJ EC01434
SMOVL C01435 BC01435 V=166.7 PL=0  +MOVJ EC01435
ARCON
SMOVL C01436 BC01436 V=8.3  +MOVJ EC01436
SMOVL C01437 BC01437 V=8.3  +MOVJ EC01437
SMOVL C01438 BC01438 V=8.3  +MOVJ EC01438
ARCOF
SMOVL C01439 BC01439 V=333.3  +MOVJ EC01439
SFTOF3D
MOVL C01440 BC01440 V=1000.0  +MOVJ EC01440 VJ=100.00
MOVJ C01441 BC01441 VJ=100.00  +MOVJ EC01441 VJ=100.00
MOVJ C01442 BC01442 VJ=100.00  +MOVJ EC01442 VJ=100.00
'cut_wire_dol
'cut_wire_dol
'cut_wire_dol
CALL JOB:CLEAN-R1_KM_3P
MOVJ C01443 BC01443 VJ=100.00  +MOVJ EC01443 VJ=100.00
MOVJ C01444 BC01444 VJ=100.00  +MOVJ EC01444 VJ=100.00
MOVJ C01445 BC01445 VJ=100.00  +MOVJ EC01445 VJ=100.00
'Path S4011
SFTOF3D
MOVJ C01446 BC01446 VJ=100.00  +MOVJ EC01446 VJ=100.00
MOVL C01447 BC01447 V=666.7  +MOVJ EC01447 VJ=100.00
SMOVL C01448 BC01448 V=166.7  +MOVJ EC01448
SREFP 3 C01449 BC01449  +REFP EC01449
CALL JOB:SEARCH-R1-S13D
SET P049 P006
SFTON3D P049
SMOVL C01450 BC01450 V=166.7  +MOVJ EC01450
SMOVL C01451 BC01451 V=166.7  +MOVJ EC01451
SREFP 3 C01452 BC01452  +REFP EC01452
CALL JOB:SEARCH-R1-S13D
SET P049 P006
SFTON3D P049
SMOVL C01453 BC01453 V=166.7  +MOVJ EC01453
SMOVL C01454 BC01454 V=166.7  +MOVJ EC01454
SMOVL C01455 BC01455 V=166.7  +MOVJ EC01455
SREFP 3 C01456 BC01456  +REFP EC01456
CALL JOB:SEARCH-R1-S13D
SET P049 P006
SFTON3D P049
SMOVL C01457 BC01457 V=166.7  +MOVJ EC01457
MOVL C01458 BC01458 V=1000.0  +MOVJ EC01458 VJ=100.00
'EndPath S4011
'Path S4010
SFTOF3D
MOVJ C01459 BC01459 VJ=100.00  +MOVJ EC01459 VJ=100.00
SMOVL C01460 BC01460 V=666.7  +MOVJ EC01460
SMOVL C01461 BC01461 V=166.7  +MOVJ EC01461
SREFP 3 C01462 BC01462  +REFP EC01462
CALL JOB:SEARCH-R1-S13D
SET P048 P006
SFTON3D P048
SMOVL C01463 BC01463 V=166.7  +MOVJ EC01463
SMOVL C01464 BC01464 V=166.7  +MOVJ EC01464
SREFP 3 C01465 BC01465  +REFP EC01465
CALL JOB:SEARCH-R1-S13D
SET P048 P006
SFTON3D P048
SMOVL C01466 BC01466 V=233.3  +MOVJ EC01466
MOVL C01467 BC01467 V=1000.0  +MOVJ EC01467 VJ=100.00
'EndPath S4010
'Path S4009
SFTOF3D
MOVJ C01468 BC01468 VJ=100.00  +MOVJ EC01468 VJ=100.00
MOVL C01469 BC01469 V=666.7  +MOVJ EC01469 VJ=100.00
SMOVL C01470 BC01470 V=166.7  +MOVJ EC01470
SREFP 3 C01471 BC01471  +REFP EC01471
CALL JOB:SEARCH-R1-S13D
SET P047 P006
SFTON3D P047
SMOVL C01472 BC01472 V=166.7  +MOVJ EC01472
SMOVL C01473 BC01473 V=166.7  +MOVJ EC01473
SREFP 3 C01474 BC01474  +REFP EC01474
CALL JOB:SEARCH-R1-S13D
SET P047 P006
SFTON3D P047
SMOVL C01475 BC01475 V=166.7  +MOVJ EC01475
MOVL C01476 BC01476 V=1000.0  +MOVJ EC01476 VJ=100.00
'EndPath S4009
MOVJ C01477 BC01477 VJ=100.00  +MOVJ EC01477 VJ=100.00
'Path S4008
SFTOF3D
MOVJ C01478 BC01478 VJ=100.00  +MOVJ EC01478 VJ=100.00
MOVL C01479 BC01479 V=666.7  +MOVJ EC01479 VJ=100.00
SMOVL C01480 BC01480 V=166.7  +MOVJ EC01480
SREFP 3 C01481 BC01481  +REFP EC01481
CALL JOB:SEARCH-R1-S13D
SET P046 P006
SFTON3D P046
SMOVL C01482 BC01482 V=166.7  +MOVJ EC01482
SMOVL C01483 BC01483 V=166.7  +MOVJ EC01483
SREFP 3 C01484 BC01484  +REFP EC01484
CALL JOB:SEARCH-R1-S13D
SET P046 P006
SFTON3D P046
SMOVL C01485 BC01485 V=166.7  +MOVJ EC01485
MOVL C01486 BC01486 V=1000.0  +MOVJ EC01486 VJ=100.00
'EndPath S4008
'Path S4007
SFTOF3D
MOVJ C01487 BC01487 VJ=100.00  +MOVJ EC01487 VJ=100.00
MOVL C01488 BC01488 V=666.7  +MOVJ EC01488 VJ=100.00
SMOVL C01489 BC01489 V=166.7  +MOVJ EC01489
SREFP 3 C01490 BC01490  +REFP EC01490
CALL JOB:SEARCH-R1-S13D
SET P055 P006
SFTON3D P055
SMOVL C01491 BC01491 V=166.7  +MOVJ EC01491
SMOVL C01492 BC01492 V=166.7  +MOVJ EC01492
SMOVL C01493 BC01493 V=166.7  +MOVJ EC01493
SREFP 3 C01494 BC01494  +REFP EC01494
CALL JOB:SEARCH-R1-S13D
SET P055 P006
SFTON3D P055
SMOVL C01495 BC01495 V=166.7  +MOVJ EC01495
SREFP 3 C01496 BC01496  +REFP EC01496
CALL JOB:SEARCH-R1-S13D
SET P045 P006
SFTON3D P045
SMOVL C01497 BC01497 V=166.7  +MOVJ EC01497
SMOVL C01498 BC01498 V=166.7  +MOVJ EC01498
SMOVL C01499 BC01499 V=166.7  +MOVJ EC01499
SREFP 3 C01500 BC01500  +REFP EC01500
CALL JOB:SEARCH-R1-S13D
SET P045 P006
SFTON3D P045
SMOVL C01501 BC01501 V=166.7  +MOVJ EC01501
MOVL C01502 BC01502 V=1000.0  +MOVJ EC01502 VJ=100.00
'EndPath S4007
'Path S3506
SFTOF3D
MOVJ C01503 BC01503 VJ=100.00  +MOVJ EC01503 VJ=100.00
MOVL C01504 BC01504 V=666.7  +MOVJ EC01504 VJ=100.00
MOVL C01505 BC01505 V=166.7  +MOVJ EC01505 VJ=0.78
SREFP 3 C01506 BC01506  +REFP EC01506
CALL JOB:SEARCH-R1-S13D
SET P054 P006
SFTON3D P054
SMOVL C01507 BC01507 V=166.7  +MOVJ EC01507
SMOVL C01508 BC01508 V=166.7  +MOVJ EC01508
SMOVL C01509 BC01509 V=166.7  +MOVJ EC01509
SREFP 3 C01510 BC01510  +REFP EC01510
CALL JOB:SEARCH-R1-S13D
SET P054 P006
SFTON3D P054
SMOVL C01511 BC01511 V=166.7  +MOVJ EC01511
SREFP 3 C01512 BC01512  +REFP EC01512
CALL JOB:SEARCH-R1-S13D
SET P044 P006
SFTON3D P044
SMOVL C01513 BC01513 V=166.7  +MOVJ EC01513
SMOVL C01514 BC01514 V=166.7  +MOVJ EC01514
SMOVL C01515 BC01515 V=166.7  +MOVJ EC01515
SREFP 3 C01516 BC01516  +REFP EC01516
CALL JOB:SEARCH-R1-S13D
SET P044 P006
SFTON3D P044
SMOVL C01517 BC01517 V=166.7  +MOVJ EC01517
MOVL C01518 BC01518 V=1000.0  +MOVJ EC01518 VJ=100.00
SFTOF3D
'EndPath S3506
MOVJ C01519 BC01519 VJ=100.00  +MOVJ EC01519 VJ=100.00
MOVJ C01520 BC01520 VJ=100.00  +MOVJ EC01520 VJ=100.00
MOVJ C01521 BC01521 VJ=100.00  +MOVJ EC01521 VJ=100.00
MOVJ C01522 BC01522 VJ=100.00  +MOVJ EC01522 VJ=100.00
MOVJ C01523 BC01523 VJ=100.00  +MOVJ EC01523 VJ=100.00
'Path S4006
SFTOF3D
MOVJ C01524 BC01524 VJ=100.00  +MOVJ EC01524 VJ=100.00
MOVL C01525 BC01525 V=666.7  +MOVJ EC01525 VJ=100.00
SMOVL C01526 BC01526 V=166.7  +MOVJ EC01526
SREFP 3 C01527 BC01527  +REFP EC01527
CALL JOB:SEARCH-R1-S13D
SET P053 P006
SFTON3D P053
SMOVL C01528 BC01528 V=166.7  +MOVJ EC01528
SMOVL C01529 BC01529 V=166.7  +MOVJ EC01529
SMOVL C01530 BC01530 V=166.7  +MOVJ EC01530
SREFP 3 C01531 BC01531  +REFP EC01531
CALL JOB:SEARCH-R1-S13D
SET P053 P006
SFTON3D P053
SMOVL C01532 BC01532 V=166.7  +MOVJ EC01532
SREFP 3 C01533 BC01533  +REFP EC01533
CALL JOB:SEARCH-R1-S13D
SET P043 P006
SFTON3D P043
SMOVL C01534 BC01534 V=166.7  +MOVJ EC01534
SMOVL C01535 BC01535 V=166.7  +MOVJ EC01535
SMOVL C01536 BC01536 V=166.7  +MOVJ EC01536
SREFP 3 C01537 BC01537  +REFP EC01537
CALL JOB:SEARCH-R1-S13D
SET P043 P006
SFTON3D P043
SMOVL C01538 BC01538 V=166.7  +MOVJ EC01538
MOVL C01539 BC01539 V=1000.0  +MOVJ EC01539 VJ=100.00
'EndPath S4006
'Path S4005
SFTOF3D
MOVJ C01540 BC01540 VJ=100.00  +MOVJ EC01540 VJ=100.00
MOVL C01541 BC01541 V=800.0  +MOVJ EC01541 VJ=100.00
SMOVL C01542 BC01542 V=166.7  +MOVJ EC01542
SREFP 3 C01543 BC01543  +REFP EC01543
CALL JOB:SEARCH-R1-S13D
SET P052 P006
SFTON3D P052
SMOVL C01544 BC01544 V=166.7  +MOVJ EC01544
SMOVL C01545 BC01545 V=166.7  +MOVJ EC01545
SMOVL C01546 BC01546 V=166.7  +MOVJ EC01546
SREFP 3 C01547 BC01547  +REFP EC01547
CALL JOB:SEARCH-R1-S13D
SET P052 P006
SFTON3D P052
SMOVL C01548 BC01548 V=166.7  +MOVJ EC01548
SREFP 3 C01549 BC01549  +REFP EC01549
CALL JOB:SEARCH-R1-S13D
SET P042 P006
SFTON3D P042
SMOVL C01550 BC01550 V=166.7  +MOVJ EC01550
SMOVL C01551 BC01551 V=166.7  +MOVJ EC01551
SMOVL C01552 BC01552 V=166.7  +MOVJ EC01552
SREFP 3 C01553 BC01553  +REFP EC01553
CALL JOB:SEARCH-R1-S13D
SET P042 P006
SFTON3D P042
SMOVL C01554 BC01554 V=166.7  +MOVJ EC01554
MOVL C01555 BC01555 V=1000.0  +MOVJ EC01555 VJ=100.00
'EndPath S4005
'Path S4004
SFTOF3D
MOVJ C01556 BC01556 VJ=100.00  +MOVJ EC01556 VJ=100.00
MOVL C01557 BC01557 V=800.0  +MOVJ EC01557 VJ=100.00
SMOVL C01558 BC01558 V=166.7  +MOVJ EC01558
SMOVL C01559 BC01559 V=166.7  +MOVJ EC01559
SREFP 3 C01560 BC01560  +REFP EC01560
CALL JOB:SEARCH-R1-S13D
SET P041 P006
SFTON3D P041
SMOVL C01561 BC01561 V=166.7  +MOVJ EC01561
SMOVL C01562 BC01562 V=166.7  +MOVJ EC01562
SREFP 3 C01563 BC01563  +REFP EC01563
CALL JOB:SEARCH-R1-S13D
SET P041 P006
SFTON3D P041
SMOVL C01564 BC01564 V=166.7  +MOVJ EC01564
SREFP 3 C01565 BC01565  +REFP EC01565
CALL JOB:SEARCH-R1-S13D
SET P041 P006
SFTON3D P041
SMOVL C01566 BC01566 V=166.7  +MOVJ EC01566
MOVL C01567 BC01567 V=1000.0  +MOVJ EC01567 VJ=100.00
'EndPath S4004
'Path S4003
SFTOF3D
MOVJ C01568 BC01568 VJ=100.00  +MOVJ EC01568 VJ=100.00
MOVL C01569 BC01569 V=800.0  +MOVJ EC01569 VJ=100.00
SMOVL C01570 BC01570 V=166.7  +MOVJ EC01570
SREFP 3 C01571 BC01571  +REFP EC01571
CALL JOB:SEARCH-R1-S13D
SET P040 P006
SFTON3D P040
SMOVL C01572 BC01572 V=250.0  +MOVJ EC01572
SMOVL C01573 BC01573 V=250.0  +MOVJ EC01573
SMOVL C01574 BC01574 V=166.7  +MOVJ EC01574
SREFP 3 C01575 BC01575  +REFP EC01575
CALL JOB:SEARCH-R1-S13D
SET P040 P006
SFTON3D P040
SMOVL C01576 BC01576 V=166.7  +MOVJ EC01576
SMOVL C01577 BC01577 V=166.7  +MOVJ EC01577
SREFP 3 C01578 BC01578  +REFP EC01578
CALL JOB:SEARCH-R1-S13D
SET P040 P006
SFTON3D P040
SMOVL C01579 BC01579 V=166.7  +MOVJ EC01579
MOVL C01580 BC01580 V=1000.0  +MOVJ EC01580 VJ=100.00
'EndPath S4003
'Path W4012
SFTOF3D
SFTON3D P040
MOVJ C01581 BC01581 VJ=100.00  +MOVJ EC01581 VJ=100.00
SMOVL C01582 BC01582 V=800.0  +MOVJ EC01582
SMOVL C01583 BC01583 V=150.0 PL=0  +MOVJ EC01583
ARCON
SMOVL C01584 BC01584 V=11.7  +MOVJ EC01584
ARCOF
SMOVL C01585 BC01585 V=800.0  +MOVJ EC01585
SMOVL C01586 BC01586 V=1000.0  +MOVJ EC01586
SFTOF3D
'EndPath W4012
'Path W4013
SFTOF3D
SFTON3D P040
MOVJ C01587 BC01587 VJ=100.00  +MOVJ EC01587 VJ=100.00
SMOVL C01588 BC01588 V=800.0  +MOVJ EC01588
SMOVL C01589 BC01589 V=150.0 PL=0  +MOVJ EC01589
ARCON
SMOVL C01590 BC01590 V=10.0  +MOVJ EC01590
ARCOF
SMOVL C01591 BC01591 V=800.0  +MOVJ EC01591
SMOVL C01592 BC01592 V=1000.0  +MOVJ EC01592
SMOVL C01593 BC01593 V=1000.0  +MOVJ EC01593
SFTOF3D
'EndPath W4013
'Path W4014
SFTOF3D
SFTON3D P040
MOVJ C01594 BC01594 VJ=100.00  +MOVJ EC01594 VJ=100.00
SMOVL C01595 BC01595 V=800.0  +MOVJ EC01595
SMOVL C01596 BC01596 V=150.0 PL=0  +MOVJ EC01596
ARCON
SMOVL C01597 BC01597 V=10.0  +MOVJ EC01597
ARCOF
SMOVL C01598 BC01598 V=800.0  +MOVJ EC01598
SMOVL C01599 BC01599 V=1000.0  +MOVJ EC01599
SFTOF3D
'EndPath W4014
'
MOVJ C01600 BC01600 VJ=100.00  +MOVJ EC01600 VJ=100.00
MOVJ C01601 BC01601 VJ=100.00  +MOVJ EC01601 VJ=100.00
MOVJ C01602 BC01602 VJ=100.00  +MOVJ EC01602 VJ=100.00
MOVJ C01603 BC01603 VJ=100.00  +MOVJ EC01603 VJ=100.00
MOVJ C01604 BC01604 VJ=100.00  +MOVJ EC01604 VJ=100.00
'Path W3522
SFTOF3D
SFTON3D P045
MOVJ C01605 BC01605 VJ=100.00  +MOVJ EC01605 VJ=100.00
SMOVL C01606 BC01606 V=800.0  +MOVJ EC01606
SMOVL C01607 BC01607 V=150.0 PL=0  +MOVJ EC01607
MACRO1 MJ#(0) ARGF9
ARCON
SMOVL C01608 BC01608 V=11.7  +MOVJ EC01608
ARCOF
SMOVL C01609 BC01609 V=800.0  +MOVJ EC01609
SMOVL C01610 BC01610 V=1000.0  +MOVJ EC01610
SFTOF3D
'EndPath W3522
'Path W3520
SFTOF3D
SFTON3D P044
MOVJ C01611 BC01611 VJ=100.00  +MOVJ EC01611 VJ=100.00
SMOVL C01612 BC01612 V=800.0  +MOVJ EC01612
SMOVL C01613 BC01613 V=166.7 PL=0  +MOVJ EC01613
ARCON
SMOVL C01614 BC01614 V=11.7  +MOVJ EC01614
SMOVL C01615 BC01615 V=11.7  +MOVJ EC01615
SMOVL C01616 BC01616 V=11.7  +MOVJ EC01616
ARCOF
SMOVL C01617 BC01617 V=800.0  +MOVJ EC01617
SMOVL C01618 BC01618 V=1000.0  +MOVJ EC01618
SFTOF3D
'EndPath W3520
'Path W3519
SFTOF3D
SFTON3D P046
MOVJ C01619 BC01619 VJ=100.00  +MOVJ EC01619 VJ=100.00
SMOVL C01620 BC01620 V=800.0  +MOVJ EC01620
SMOVL C01621 BC01621 V=166.7 PL=0  +MOVJ EC01621
ARCON
SMOVL C01622 BC01622 V=12.5  +MOVJ EC01622
SMOVL C01623 BC01623 V=12.5  +MOVJ EC01623
SMOVL C01624 BC01624 V=12.5  +MOVJ EC01624
ARCOF
SMOVL C01625 BC01625 V=800.0  +MOVJ EC01625
SMOVL C01626 BC01626 V=1000.0  +MOVJ EC01626
SFTOF3D
'EndPath W3519
'1
MOVJ C01627 BC01627 VJ=100.00  +MOVJ EC01627 VJ=100.00
MOVJ C01628 BC01628 VJ=100.00  +MOVJ EC01628 VJ=100.00
'Path W3509
SFTOF3D
SFTON3D P048
MOVJ C01629 BC01629 VJ=100.00  +MOVJ EC01629 VJ=100.00
SMOVL C01630 BC01630 V=800.0  +MOVJ EC01630
SMOVL C01631 BC01631 V=150.0 PL=0  +MOVJ EC01631
ARCON
SMOVL C01632 BC01632 V=11.7  +MOVJ EC01632
ARCOF
SMOVL C01633 BC01633 V=800.0  +MOVJ EC01633
SMOVL C01634 BC01634 V=1000.0  +MOVJ EC01634
SFTOF3D
'EndPath W3509
'Path W3510
SFTOF3D
SFTON3D P049
MOVJ C01635 BC01635 VJ=100.00  +MOVJ EC01635 VJ=100.00
SMOVL C01636 BC01636 V=800.0  +MOVJ EC01636
SMOVL C01637 BC01637 V=150.0 PL=0  +MOVJ EC01637
MACRO1 MJ#(0) ARGF6
ARCON
SMOVL C01638 BC01638 V=9.2  +MOVJ EC01638
SMOVL C01639 BC01639 V=9.2  +MOVJ EC01639
SMOVL C01640 BC01640 V=9.2  +MOVJ EC01640
SMOVL C01641 BC01641 V=9.2  +MOVJ EC01641
SMOVL C01642 BC01642 V=9.2  +MOVJ EC01642
ARCOF
MOVJ C01643 BC01643 VJ=30.00  +MOVJ EC01643 VJ=80.00
MOVJ C01644 BC01644 VJ=30.00  +MOVJ EC01644 VJ=30.00
SMOVL C01645 BC01645 V=166.7  +MOVJ EC01645
ARCON
SMOVL C01646 BC01646 V=13.3  +MOVJ EC01646
SMOVL C01647 BC01647 V=13.3  +MOVJ EC01647
SMOVL C01648 BC01648 V=13.3  +MOVJ EC01648
ARCOF
SMOVL C01649 BC01649 V=333.3  +MOVJ EC01649
SMOVL C01650 BC01650 V=666.7  +MOVJ EC01650
SMOVL C01651 BC01651 V=166.7  +MOVJ EC01651
ARCON
SMOVL C01652 BC01652 V=13.3  +MOVJ EC01652
SMOVL C01653 BC01653 V=13.3  +MOVJ EC01653
ARCOF
SMOVL C01654 BC01654 V=166.7  +MOVJ EC01654
ARCON
SMOVL C01655 BC01655 V=11.7  +MOVJ EC01655
ARCOF
SMOVL C01656 BC01656 V=250.0  +MOVJ EC01656
SFTOF3D
'EndPath W3510
MOVJ C01657 BC01657 VJ=100.00  +MOVJ EC01657 VJ=100.00
'2
MOVJ C01658 BC01658 VJ=100.00  +MOVJ EC01658 VJ=100.00
MOVJ C01659 BC01659 VJ=100.00  +MOVJ EC01659 VJ=100.00
MOVJ C01660 BC01660 VJ=100.00  +MOVJ EC01660 VJ=100.00
'Path W3511
SFTOF3D
SFTON3D P043
MOVJ C01661 BC01661 VJ=100.00  +MOVJ EC01661 VJ=100.00
SMOVL C01662 BC01662 V=800.0  +MOVJ EC01662
SMOVL C01663 BC01663 V=166.7 PL=0  +MOVJ EC01663
MACRO1 MJ#(0) ARGF9
ARCON
SMOVL C01664 BC01664 V=11.7  +MOVJ EC01664
ARCOF
SMOVL C01665 BC01665 V=800.0  +MOVJ EC01665
SMOVL C01666 BC01666 V=1000.0  +MOVJ EC01666
SFTOF3D
'EndPath W3511
'Path W3512
SFTOF3D
SFTON3D P042
MOVJ C01667 BC01667 VJ=100.00  +MOVJ EC01667 VJ=100.00
SMOVL C01668 BC01668 V=800.0  +MOVJ EC01668
SMOVL C01669 BC01669 V=150.0 PL=0  +MOVJ EC01669
ARCON
SMOVL C01670 BC01670 V=11.7  +MOVJ EC01670
ARCOF
SMOVL C01671 BC01671 V=800.0  +MOVJ EC01671
SMOVL C01672 BC01672 V=1000.0  +MOVJ EC01672
SFTOF3D
'EndPath W3512
'3
MOVJ C01673 BC01673 VJ=100.00  +MOVJ EC01673 VJ=100.00
MOVJ C01674 BC01674 VJ=100.00  +MOVJ EC01674 VJ=100.00
MOVJ C01675 BC01675 VJ=100.00  +MOVJ EC01675 VJ=100.00
MOVJ C01676 BC01676 VJ=100.00  +MOVJ EC01676 VJ=100.00
'Path W3514
SFTOF3D
SFTON3D P047
MOVJ C01677 BC01677 VJ=100.00  +MOVJ EC01677 VJ=100.00
SMOVL C01678 BC01678 V=800.0  +MOVJ EC01678
SMOVL C01679 BC01679 V=150.0 PL=0  +MOVJ EC01679
ARCON
SMOVL C01680 BC01680 V=11.7  +MOVJ EC01680
ARCOF
SMOVL C01681 BC01681 V=800.0  +MOVJ EC01681
SMOVL C01682 BC01682 V=1000.0  +MOVJ EC01682
SFTOF3D
'EndPath W3514
'Path W3518
SFTOF3D
SFTON3D P047
MOVJ C01683 BC01683 VJ=100.00  +MOVJ EC01683 VJ=100.00
SMOVL C01684 BC01684 V=800.0  +MOVJ EC01684
SMOVL C01685 BC01685 V=150.0 PL=0  +MOVJ EC01685
ARCON
SMOVL C01686 BC01686 V=11.7  +MOVJ EC01686
ARCOF
SMOVL C01687 BC01687 V=800.0  +MOVJ EC01687
SMOVL C01688 BC01688 V=1000.0  +MOVJ EC01688
SFTOF3D
'EndPath W3518
MOVJ C01689 BC01689 VJ=100.00  +MOVJ EC01689 VJ=100.00
MOVJ C01690 BC01690 VJ=100.00  +MOVJ EC01690 VJ=100.00
MOVJ C01691 BC01691 VJ=100.00  +MOVJ EC01691 VJ=100.00
MOVJ C01692 BC01692 VJ=100.00  +MOVJ EC01692 VJ=100.00
'Path W3516
SFTOF3D
SFTON3D P043
MOVJ C01693 BC01693 VJ=50.00  +MOVJ EC01693 VJ=50.00
MOVJ C01694 BC01694 VJ=100.00  +MOVJ EC01694 VJ=100.00
SMOVL C01695 BC01695 V=800.0  +MOVJ EC01695
SMOVL C01696 BC01696 V=150.0 PL=0  +MOVJ EC01696
ARCON
SMOVL C01697 BC01697 V=11.7  +MOVJ EC01697
ARCOF
SMOVL C01698 BC01698 V=800.0  +MOVJ EC01698
SMOVL C01699 BC01699 V=1000.0  +MOVJ EC01699
SFTOF3D
'EndPath W3516
'Path W3515
SFTOF3D
SFTON3D P042
MOVJ C01700 BC01700 VJ=100.00  +MOVJ EC01700 VJ=100.00
SMOVL C01701 BC01701 V=800.0  +MOVJ EC01701
SMOVL C01702 BC01702 V=166.7 PL=0  +MOVJ EC01702
ARCON
SMOVL C01703 BC01703 V=10.8  +MOVJ EC01703
ARCOF
SMOVL C01704 BC01704 V=800.0  +MOVJ EC01704
SMOVL C01705 BC01705 V=1000.0  +MOVJ EC01705
SFTOF3D
'EndPath W3515
MOVJ C01706 BC01706 VJ=100.00  +MOVJ EC01706 VJ=100.00
MOVJ C01707 BC01707 VJ=100.00  +MOVJ EC01707 VJ=100.00
MOVJ C01708 BC01708 VJ=100.00  +MOVJ EC01708 VJ=100.00
MOVJ C01709 BC01709 VJ=100.00  +MOVJ EC01709 VJ=100.00
'Path W3523
SFTOF3D
SFTON3D P046
MOVJ C01710 BC01710 VJ=100.00  +MOVJ EC01710 VJ=100.00
SMOVL C01711 BC01711 V=800.0  +MOVJ EC01711
SMOVL C01712 BC01712 V=166.7 PL=0  +MOVJ EC01712
MACRO1 MJ#(0) ARGF14
ARCON
SMOVL C01713 BC01713 V=10.0  +MOVJ EC01713
ARCOF
SMOVL C01714 BC01714 V=800.0  +MOVJ EC01714
SMOVL C01715 BC01715 V=1000.0  +MOVJ EC01715
SFTOF3D
'EndPath W3523
'Path W4015
SFTOF3D
SFTON3D P044
MOVJ C01716 BC01716 VJ=100.00  +MOVJ EC01716 VJ=100.00
SMOVL C01717 BC01717 V=800.0  +MOVJ EC01717
SMOVL C01718 BC01718 V=150.0 PL=0  +MOVJ EC01718
MACRO1 MJ#(0) ARGF9
ARCON
SMOVL C01719 BC01719 V=10.8  +MOVJ EC01719
ARCOF
SMOVL C01720 BC01720 V=800.0  +MOVJ EC01720
SMOVL C01721 BC01721 V=1000.0  +MOVJ EC01721
SFTOF3D
'EndPath W4015
MOVJ C01722 BC01722 VJ=100.00  +MOVJ EC01722 VJ=100.00
MOVJ C01723 BC01723 VJ=100.00  +MOVJ EC01723 VJ=100.00
MOVJ C01724 BC01724 VJ=100.00  +MOVJ EC01724 VJ=100.00
MOVJ C01725 BC01725 VJ=100.00  +MOVJ EC01725 VJ=100.00
'Path W4016
SFTOF3D
SFTON3D P041
MOVJ C01726 BC01726 VJ=100.00  +MOVJ EC01726 VJ=100.00
SMOVL C01727 BC01727 V=800.0  +MOVJ EC01727
SMOVL C01728 BC01728 V=150.0 PL=0  +MOVJ EC01728
MACRO1 MJ#(0) ARGF14
ARCON
SMOVL C01729 BC01729 V=10.0  +MOVJ EC01729
SMOVL C01730 BC01730 V=10.0  +MOVJ EC01730
SMOVL C01731 BC01731 V=10.0  +MOVJ EC01731
ARCOF
SMOVL C01732 BC01732 V=800.0  +MOVJ EC01732
SMOVL C01733 BC01733 V=1000.0  +MOVJ EC01733
SFTOF3D
COMM 'EndPath W4016
COMM 'Path W4017
COMM SFTOF3D
COMM SFTON3D P041
COMM MOVJ C01734 BC01734 VJ=100.00  +MOVJ EC01734 VJ=100.00
COMM SMOVL C01735 BC01735 V=800.0  +MOVJ EC01735
COMM SMOVL C01736 BC01736 V=150.0 PL=0  +MOVJ EC01736
COMM SMOVL C01737 BC01737 V=10.0  +MOVJ EC01737
COMM ARCOF
COMM SMOVL C01738 BC01738 V=800.0  +MOVJ EC01738
COMM SMOVL C01739 BC01739 V=1000.0  +MOVJ EC01739
COMM SFTOF3D
COMM 'EndPath W4017
COMM MOVJ C01740 BC01740 VJ=100.00  +MOVJ EC01740 VJ=100.00
COMM 'Path W4018
COMM SFTOF3D
COMM SFTON3D P041
COMM MOVJ C01741 BC01741 VJ=100.00  +MOVJ EC01741 VJ=100.00
COMM SMOVL C01742 BC01742 V=800.0  +MOVJ EC01742
COMM SMOVL C01743 BC01743 V=150.0 PL=0  +MOVJ EC01743
COMM SMOVL C01744 BC01744 V=10.0  +MOVJ EC01744
COMM ARCOF
COMM SMOVL C01745 BC01745 V=800.0  +MOVJ EC01745
COMM SMOVL C01746 BC01746 V=1000.0  +MOVJ EC01746
COMM SFTOF3D
'EndPath W4018
MOVJ C01747 BC01747 VJ=100.00  +MOVJ EC01747 VJ=100.00
MOVJ C01748 BC01748 VJ=100.00  +MOVJ EC01748 VJ=100.00
MOVJ C01749 BC01749 VJ=100.00  +MOVJ EC01749 VJ=100.00
MOVJ C01750 BC01750 VJ=100.00  +MOVJ EC01750 VJ=100.00
MOVJ C01751 BC01751 VJ=100.00  +MOVJ EC01751 VJ=100.00
END
